C07270=1079.126,-46.331,-56.939,173.614,20.204,153.491
C07271=1079.132,-46.080,-56.951,173.616,20.206,153.491
C07272=1079.137,-45.831,-56.963,173.617,20.207,153.491
C07273=1079.144,-45.582,-56.975,173.618,20.209,153.491
C07274=1079.150,-45.332,-56.987,173.621,20.212,153.491
C07275=1079.155,-45.083,-57.000,173.622,20.214,153.492
C07276=1079.162,-44.833,-57.012,173.623,20.215,153.492
C07277=1079.168,-44.583,-57.024,173.625,20.217,153.492
C07278=1079.173,-44.334,-57.035,173.626,20.219,153.492
C07279=1079.179,-44.084,-57.048,173.627,20.221,153.492
C07280=1079.185,-43.834,-57.060,173.629,20.223,153.492
C07281=1079.192,-43.584,-57.072,173.630,20.225,153.492
C07282=1079.197,-43.335,-57.084,173.632,20.227,153.492
C07283=1079.203,-43.085,-57.097,173.633,20.229,153.493
C07284=1079.210,-42.836,-57.109,173.635,20.230,153.493
C07285=1079.215,-42.586,-57.121,173.636,20.232,153.493
C07286=1079.221,-42.337,-57.134,173.637,20.234,153.493
C07287=1079.228,-42.087,-57.146,173.639,20.236,153.493
C07288=1079.233,-41.837,-57.158,173.640,20.238,153.493
C07289=1079.239,-41.588,-57.170,173.642,20.240,153.493
C07290=1079.245,-41.338,-57.183,173.644,20.242,153.493
C07291=1079.251,-41.088,-57.195,173.645,20.244,153.494
C07292=1079.257,-40.839,-57.207,173.646,20.246,153.494
C07293=1079.263,-40.589,-57.220,173.648,20.248,153.494
C07294=1079.269,-40.340,-57.231,173.649,20.250,153.494
C07295=1079.275,-40.090,-57.244,173.650,20.252,153.494
C07296=1079.281,-39.840,-57.257,173.652,20.253,153.494
C07297=1079.288,-39.590,-57.269,173.653,20.255,153.494
C07298=1079.293,-39.341,-57.281,173.655,20.258,153.494
C07299=1079.299,-39.091,-57.293,173.657,20.260,153.495
C07300=1079.305,-38.842,-57.306,173.658,20.262,153.495
C07301=1079.311,-38.592,-57.318,173.659,20.263,153.495
C07302=1079.317,-38.342,-57.330,173.661,20.265,153.495
C07303=1079.323,-38.093,-57.343,173.662,20.267,153.495
C07304=1079.329,-37.843,-57.355,173.663,20.269,153.495
C07305=1079.334,-37.593,-57.368,173.665,20.272,153.495
C07306=1079.340,-37.343,-57.380,173.667,20.274,153.496
C07307=1079.346,-37.094,-57.392,173.668,20.276,153.496
C07308=1079.353,-36.845,-57.405,173.669,20.278,153.496
C07309=1079.359,-36.595,-57.418,173.671,20.279,153.496
C07310=1079.364,-36.345,-57.430,173.672,20.281,153.496
C07311=1079.370,-36.096,-57.442,173.673,20.283,153.496
C07312=1079.376,-35.846,-57.455,173.674,20.285,153.496
C07313=1079.382,-35.596,-57.467,173.677,20.288,153.497
C07314=1079.388,-35.347,-57.480,173.678,20.290,153.497
C07315=1079.393,-35.097,-57.493,173.679,20.292,153.497
C07316=1079.399,-34.848,-57.505,173.680,20.294,153.497
C07317=1079.406,-34.599,-57.517,173.682,20.296,153.497
C07318=1079.412,-34.349,-57.530,173.683,20.298,153.497
C07319=1079.417,-34.099,-57.543,173.685,20.300,153.497
C07320=1079.423,-33.849,-57.555,173.687,20.302,153.498
C07321=1079.430,-33.575,-57.569,173.688,20.304,153.498
C07322=1079.436,-33.302,-57.583,173.689,20.306,153.498
C07323=1079.442,-33.028,-57.596,173.691,20.309,153.498
C07324=1079.449,-32.754,-57.610,173.692,20.311,153.498
C07325=1079.455,-32.504,-57.624,173.694,20.313,153.499
C07326=1079.461,-32.254,-57.636,173.695,20.315,153.499
C07327=1079.467,-32.004,-57.649,173.697,20.317,153.499
C07328=1079.473,-31.755,-57.661,173.699,20.318,153.499
C07329=1079.479,-31.505,-57.675,173.700,20.320,153.499
C07330=1079.484,-31.256,-57.687,173.701,20.322,153.499
C07331=1079.491,-31.007,-57.699,173.703,20.324,153.499
C07332=1079.497,-30.757,-57.712,173.704,20.326,153.500
C07333=1079.503,-30.507,-57.725,173.705,20.328,153.500
C07334=1079.509,-30.258,-57.737,173.707,20.331,153.500
C07335=1079.515,-30.008,-57.750,173.709,20.333,153.500
C07336=1079.521,-29.758,-57.763,173.710,20.335,153.500
C07337=1079.527,-29.509,-57.775,173.711,20.337,153.500
C07338=1079.532,-29.259,-57.788,173.712,20.339,153.500
C07339=1079.538,-29.010,-57.801,173.714,20.341,153.501
C07340=1079.544,-28.760,-57.813,173.716,20.343,153.501
C07341=1079.550,-28.510,-57.826,173.717,20.345,153.501
C07342=1079.556,-28.261,-57.839,173.719,20.347,153.501
C07343=1079.562,-28.011,-57.852,173.720,20.349,153.501
C07344=1079.568,-27.761,-57.864,173.721,20.351,153.501
C07345=1079.574,-27.512,-57.878,173.722,20.353,153.501
C07346=1079.580,-27.262,-57.890,173.725,20.355,153.502
C07347=1079.587,-27.013,-57.903,173.726,20.357,153.502
C07348=1079.592,-26.763,-57.916,173.727,20.359,153.502
C07349=1079.598,-26.513,-57.929,173.728,20.361,153.502
C07350=1079.604,-26.264,-57.942,173.730,20.363,153.502
C07351=1079.609,-26.014,-57.955,173.731,20.365,153.502
C07352=1079.615,-25.765,-57.968,173.733,20.368,153.503
C07353=1079.621,-25.515,-57.980,173.734,20.370,153.503
C07354=1079.627,-25.266,-57.994,173.736,20.372,153.503
C07355=1079.633,-25.016,-58.006,173.737,20.374,153.503
C07356=1079.639,-24.766,-58.019,173.738,20.376,153.503
C07357=1079.645,-24.517,-58.033,173.739,20.378,153.504
C07358=1079.651,-24.267,-58.045,173.742,20.381,153.504
C07359=1079.657,-24.017,-58.059,173.743,20.383,153.504
C07360=1079.663,-23.768,-58.071,173.744,20.385,153.504
C07361=1079.668,-23.518,-58.085,173.745,20.387,153.504
C07362=1079.674,-23.268,-58.097,173.747,20.389,153.504
C07363=1079.680,-23.020,-58.110,173.748,20.391,153.504
C07364=1079.686,-22.770,-58.123,173.750,20.393,153.505
C07365=1079.692,-22.520,-58.136,173.751,20.395,153.505
C07366=1079.697,-22.270,-58.149,173.753,20.397,153.505
C07367=1079.703,-22.021,-58.163,173.754,20.399,153.505
C07368=1079.709,-21.771,-58.175,173.755,20.401,153.505
C07369=1079.715,-21.522,-58.188,173.757,20.403,153.505
C07370=1079.722,-21.273,-58.202,173.759,20.405,153.506
C07371=1079.727,-21.022,-58.215,173.760,20.407,153.506
C07372=1079.733,-20.773,-58.228,173.761,20.409,153.506
C07373=1079.739,-20.523,-58.241,173.763,20.411,153.506
C07374=1079.745,-20.274,-58.254,173.764,20.413,153.506
C07375=1079.751,-20.024,-58.268,173.766,20.416,153.507
C07376=1079.757,-19.774,-58.280,173.767,20.418,153.507
C07377=1079.763,-19.525,-58.294,173.768,20.420,153.507
C07378=1079.769,-19.275,-58.306,173.770,20.422,153.507
C07379=1079.774,-19.026,-58.320,173.771,20.424,153.507
C07380=1079.780,-18.776,-58.333,173.772,20.426,153.507
C07381=1079.786,-18.527,-58.346,173.774,20.429,153.507
C07382=1079.792,-18.277,-58.359,173.776,20.431,153.508
C07383=1079.798,-18.028,-58.373,173.777,20.433,153.508
C07384=1079.804,-17.778,-58.386,173.778,20.435,153.508
C07385=1079.811,-17.503,-58.400,173.780,20.437,153.508
C07386=1079.817,-17.228,-58.415,173.782,20.440,153.508
C07387=1079.824,-16.953,-58.430,173.783,20.442,153.509
C07388=1079.830,-16.679,-58.443,173.785,20.444,153.509
C07389=1079.837,-16.429,-58.457,173.786,20.446,153.509
C07390=1079.842,-16.180,-58.471,173.788,20.448,153.509
C07391=1079.849,-15.930,-58.484,173.789,20.450,153.509
C07392=1079.854,-15.680,-58.497,173.791,20.453,153.509
C07393=1079.860,-15.431,-58.511,173.792,20.455,153.510
C07394=1079.866,-15.182,-58.524,173.793,20.457,153.510
C07395=1079.872,-14.932,-58.537,173.795,20.459,153.510
C07396=1079.878,-14.682,-58.550,173.796,20.461,153.510
C07397=1079.884,-14.433,-58.564,173.797,20.463,153.510
C07398=1079.889,-14.183,-58.577,173.799,20.465,153.510
C07399=1079.895,-13.934,-58.591,173.800,20.468,153.511
C07400=1079.901,-13.684,-58.604,173.802,20.470,153.511
C07401=1079.907,-13.435,-58.617,173.803,20.472,153.511
C07402=1079.913,-13.185,-58.630,173.804,20.474,153.511
C07403=1079.919,-12.936,-58.644,173.806,20.476,153.511
C07404=1079.925,-12.686,-58.658,173.808,20.478,153.512
C07405=1079.930,-12.436,-58.671,173.809,20.481,153.512
C07406=1079.936,-12.187,-58.684,173.810,20.483,153.512
C07407=1079.942,-11.937,-58.698,173.811,20.485,153.512
C07408=1079.948,-11.687,-58.711,173.814,20.487,153.512
C07409=1079.954,-11.438,-58.725,173.815,20.489,153.512
C07410=1079.960,-11.189,-58.739,173.816,20.491,153.513
C07411=1079.965,-10.938,-58.752,173.817,20.494,153.513
C07412=1079.972,-10.689,-58.765,173.819,20.496,153.513
C07413=1079.977,-10.440,-58.779,173.821,20.498,153.513
C07414=1079.983,-10.190,-58.792,173.822,20.500,153.513
C07415=1079.989,-9.941,-58.806,173.823,20.502,153.514
C07416=1079.995,-9.691,-58.819,173.825,20.504,153.514
C07417=1080.001,-9.441,-58.834,173.826,20.507,153.514
C07418=1080.007,-9.192,-58.847,173.828,20.509,153.514
C07419=1080.013,-8.942,-58.861,173.829,20.511,153.514
C07420=1080.019,-8.693,-58.874,173.830,20.513,153.515
C07421=1080.024,-8.443,-58.887,173.832,20.515,153.515
C07422=1080.030,-8.193,-58.901,173.833,20.517,153.515
C07423=1080.036,-7.944,-58.914,173.835,20.520,153.515
C07424=1080.042,-7.694,-58.928,173.836,20.522,153.515
C07425=1080.048,-7.445,-58.942,173.837,20.524,153.515
C07426=1080.053,-7.195,-58.956,173.839,20.526,153.516
C07427=1080.060,-6.946,-58.969,173.840,20.528,153.516
C07428=1080.065,-6.696,-58.983,173.842,20.530,153.516
C07429=1080.071,-6.447,-58.996,173.843,20.533,153.516
C07430=1080.077,-6.197,-59.010,173.845,20.535,153.516
C07431=1080.084,-5.947,-59.024,173.846,20.537,153.517
C07432=1080.089,-5.698,-59.037,173.848,20.539,153.517
C07433=1080.095,-5.448,-59.051,173.849,20.541,153.517
C07434=1080.101,-5.199,-59.064,173.850,20.544,153.517
C07435=1080.107,-4.949,-59.079,173.852,20.546,153.517
C07436=1080.113,-4.699,-59.092,173.853,20.548,153.517
C07437=1080.119,-4.450,-59.106,173.855,20.550,153.518
C07438=1080.125,-4.201,-59.120,173.856,20.552,153.518
C07439=1080.131,-3.952,-59.134,173.858,20.554,153.518
C07440=1080.137,-3.701,-59.148,173.859,20.557,153.518
C07441=1080.143,-3.452,-59.161,173.860,20.559,153.518
C07442=1080.148,-3.202,-59.175,173.862,20.561,153.519
C07443=1080.154,-2.953,-59.189,173.864,20.563,153.519
C07444=1080.160,-2.704,-59.202,173.865,20.566,153.519
C07445=1080.166,-2.453,-59.216,173.866,20.568,153.519
C07446=1080.172,-2.204,-59.230,173.868,20.570,153.519
C07447=1080.177,-1.954,-59.244,173.869,20.572,153.519
C07448=1080.183,-1.705,-59.259,173.871,20.575,153.520
C07449=1080.190,-1.429,-59.273,173.872,20.577,153.520
C07450=1080.196,-1.153,-59.289,173.874,20.580,153.520
C07451=1080.202,-0.875,-59.305,173.875,20.582,153.520
C07452=1080.209,-0.600,-59.320,173.877,20.585,153.521
C07453=1080.215,-0.350,-59.334,173.878,20.587,153.521
C07454=1080.220,-0.100,-59.348,173.880,20.589,153.521
C07455=1080.226,0.148,-59.362,173.881,20.591,153.521
C07456=1080.232,0.399,-59.376,173.883,20.593,153.521
C07457=1080.237,0.648,-59.390,173.884,20.595,153.522
C07458=1080.244,0.898,-59.403,173.885,20.598,153.522
C07459=1080.249,1.147,-59.417,173.887,20.600,153.522
C07460=1080.255,1.396,-59.432,173.889,20.602,153.522
C07461=1080.261,1.646,-59.446,173.890,20.604,153.522
C07462=1080.266,1.896,-59.460,173.891,20.607,153.523
C07463=1080.272,2.146,-59.474,173.892,20.609,153.523
C07464=1080.278,2.395,-59.488,173.894,20.611,153.523
C07465=1080.284,2.644,-59.502,173.896,20.614,153.523
C07466=1080.290,2.894,-59.516,173.897,20.616,153.523
C07467=1080.296,3.143,-59.531,173.898,20.618,153.524
C07468=1080.301,3.393,-59.544,173.900,20.620,153.524
C07469=1080.307,3.643,-59.559,173.901,20.623,153.524
C07470=1080.313,3.892,-59.572,173.903,20.625,153.524
C07471=1080.319,4.141,-59.587,173.904,20.627,153.524
C07472=1080.324,4.391,-59.601,173.905,20.629,153.525
C07473=1080.331,4.641,-59.615,173.907,20.632,153.525
C07474=1080.337,4.890,-59.629,173.909,20.634,153.525
C07475=1080.342,5.139,-59.643,173.910,20.636,153.525
C07476=1080.348,5.390,-59.657,173.911,20.638,153.525
C07477=1080.354,5.639,-59.672,173.913,20.641,153.526
C07478=1080.359,5.888,-59.686,173.914,20.643,153.526
C07479=1080.366,6.138,-59.701,173.916,20.644,153.526
C07480=1080.371,6.388,-59.714,173.917,20.647,153.526
C07481=1080.377,6.637,-59.728,173.918,20.649,153.526
C07482=1080.383,6.887,-59.743,173.920,20.651,153.527
C07483=1080.389,7.136,-59.757,173.921,20.654,153.527
C07484=1080.395,7.385,-59.771,173.923,20.656,153.527
C07485=1080.401,7.635,-59.785,173.924,20.658,153.527
C07486=1080.407,7.885,-59.799,173.926,20.660,153.527
C07487=1080.413,8.134,-59.814,173.927,20.663,153.528
C07488=1080.419,8.384,-59.828,173.929,20.665,153.528
C07489=1080.424,8.633,-59.843,173.930,20.667,153.528
C07490=1080.430,8.883,-59.856,173.932,20.669,153.528
C07491=1080.436,9.132,-59.871,173.933,20.672,153.528
C07492=1080.442,9.382,-59.885,173.934,20.674,153.529
C07493=1080.447,9.631,-59.900,173.936,20.676,153.529
C07494=1080.454,9.881,-59.914,173.938,20.678,153.529
C07495=1080.459,10.130,-59.929,173.939,20.681,153.529
C07496=1080.465,10.380,-59.943,173.940,20.683,153.529
C07497=1080.471,10.629,-59.958,173.942,20.685,153.530
C07498=1080.477,10.879,-59.971,173.944,20.687,153.530
C07499=1080.483,11.128,-59.986,173.945,20.690,153.530
C07500=1080.489,11.378,-60.000,173.946,20.691,153.530
C07501=1080.496,11.627,-60.015,173.947,20.693,153.530
C07502=1080.501,11.877,-60.028,173.949,20.695,153.530
C07503=1080.508,12.127,-60.043,173.951,20.698,153.531
C07504=1080.513,12.376,-60.057,173.952,20.700,153.531
C07505=1080.519,12.625,-60.072,173.953,20.702,153.531
C07506=1080.525,12.875,-60.087,173.955,20.704,153.531
C07507=1080.531,13.124,-60.101,173.957,20.707,153.532
C07508=1080.537,13.374,-60.116,173.958,20.709,153.532
C07509=1080.542,13.624,-60.129,173.959,20.711,153.532
C07510=1080.549,13.873,-60.144,173.960,20.713,153.532
C07511=1080.555,14.122,-60.159,173.962,20.716,153.532
C07512=1080.561,14.372,-60.173,173.964,20.718,153.532
C07513=1080.566,14.650,-60.189,173.965,20.720,153.533
C07514=1080.573,14.929,-60.206,173.967,20.723,153.533
C07515=1080.579,15.207,-60.222,173.969,20.726,153.533
C07516=1080.586,15.485,-60.238,173.970,20.728,153.533
C07517=1080.592,15.735,-60.253,173.971,20.731,153.534
C07518=1080.598,15.984,-60.268,173.974,20.733,153.534
C07519=1080.604,16.234,-60.282,173.975,20.735,153.534
C07520=1080.610,16.483,-60.297,173.976,20.737,153.534
C07521=1080.615,16.732,-60.311,173.977,20.739,153.534
C07522=1080.621,16.983,-60.326,173.979,20.742,153.535
C07523=1080.626,17.232,-60.341,173.980,20.744,153.535
C07524=1080.633,17.482,-60.356,173.982,20.746,153.535
C07525=1080.639,17.730,-60.370,173.983,20.748,153.535
C07526=1080.645,17.981,-60.385,173.985,20.751,153.535
C07527=1080.650,18.230,-60.400,173.986,20.753,153.536
C07528=1080.656,18.480,-60.415,173.988,20.755,153.536
C07529=1080.662,18.729,-60.429,173.989,20.757,153.536
C07530=1080.668,18.979,-60.444,173.991,20.760,153.536
C07531=1080.674,19.228,-60.458,173.992,20.762,153.536
C07532=1080.679,19.478,-60.474,173.994,20.764,153.537
C07533=1080.685,19.727,-60.488,173.995,20.767,153.537
C07534=1080.692,19.976,-60.503,173.997,20.769,153.537
C07535=1080.697,20.226,-60.517,173.998,20.771,153.537
C07536=1080.703,20.476,-60.533,173.999,20.773,153.537
C07537=1080.708,20.725,-60.547,174.001,20.776,153.538
C07538=1080.714,20.974,-60.562,174.003,20.778,153.538
C07539=1080.720,21.224,-60.577,174.004,20.780,153.538
C07540=1080.725,21.473,-60.591,174.005,20.782,153.538
C07541=1080.732,21.723,-60.606,174.007,20.785,153.538
C07542=1080.737,21.972,-60.621,174.008,20.787,153.539
C07543=1080.743,22.222,-60.636,174.010,20.789,153.539
C07544=1080.749,22.471,-60.651,174.011,20.791,153.539
C07545=1080.755,22.721,-60.666,174.013,20.794,153.539
C07546=1080.760,22.970,-60.681,174.014,20.796,153.539
C07547=1080.767,23.220,-60.696,174.016,20.798,153.540
C07548=1080.772,23.470,-60.711,174.017,20.801,153.540
C07549=1080.778,23.719,-60.725,174.019,20.803,153.540
C07550=1080.784,23.969,-60.740,174.020,20.805,153.540
C07551=1080.789,24.218,-60.755,174.021,20.808,153.541
C07552=1080.796,24.468,-60.770,174.023,20.810,153.541
C07553=1080.801,24.717,-60.785,174.025,20.812,153.541
C07554=1080.807,24.967,-60.800,174.026,20.814,153.541
C07555=1080.813,25.216,-60.815,174.027,20.816,153.541
C07556=1080.819,25.466,-60.831,174.029,20.819,153.541
C07557=1080.824,25.714,-60.845,174.031,20.821,153.542
C07558=1080.831,25.964,-60.860,174.032,20.823,153.542
C07559=1080.836,26.214,-60.876,174.034,20.826,153.542
C07560=1080.842,26.463,-60.890,174.035,20.828,153.542
C07561=1080.849,26.713,-60.905,174.036,20.830,153.543
C07562=1080.854,26.962,-60.920,174.038,20.832,153.543
C07563=1080.860,27.212,-60.935,174.040,20.835,153.543
C07564=1080.866,27.462,-60.951,174.041,20.837,153.543
C07565=1080.871,27.711,-60.965,174.042,20.839,153.543
C07566=1080.877,27.961,-60.981,174.043,20.841,153.544
C07567=1080.883,28.209,-60.996,174.045,20.844,153.544
C07568=1080.889,28.459,-61.010,174.047,20.846,153.544
C07569=1080.895,28.708,-61.026,174.048,20.848,153.544
C07570=1080.901,28.957,-61.041,174.050,20.850,153.544
C07571=1080.907,29.207,-61.057,174.051,20.853,153.545
C07572=1080.912,29.457,-61.072,174.053,20.855,153.545
C07573=1080.918,29.706,-61.087,174.054,20.857,153.545
C07574=1080.923,29.956,-61.102,174.056,20.860,153.545
C07575=1080.929,30.205,-61.117,174.057,20.862,153.545
C07576=1080.935,30.455,-61.133,174.058,20.864,153.546
C07577=1080.941,30.735,-61.150,174.061,20.867,153.546
C07578=1080.948,31.014,-61.167,174.063,20.870,153.546
C07579=1080.954,31.294,-61.184,174.064,20.872,153.546
C07580=1080.961,31.574,-61.201,174.066,20.874,153.546
C07581=1080.967,31.823,-61.216,174.067,20.876,153.547
C07582=1080.972,32.073,-61.231,174.068,20.879,153.547
C07583=1080.978,32.321,-61.247,174.070,20.881,153.547
C07584=1080.984,32.571,-61.262,174.072,20.883,153.547
C07585=1080.990,32.821,-61.278,174.073,20.886,153.548
C07586=1080.995,33.070,-61.292,174.074,20.888,153.548
C07587=1081.001,33.320,-61.308,174.076,20.890,153.548
C07588=1081.008,33.569,-61.324,174.077,20.893,153.548
C07589=1081.013,33.818,-61.339,174.079,20.895,153.548
C07590=1081.019,34.068,-61.354,174.081,20.897,153.548
C07591=1081.025,34.318,-61.369,174.082,20.900,153.549
C07592=1081.030,34.567,-61.385,174.083,20.902,153.549
C07593=1081.037,34.816,-61.400,174.085,20.904,153.549
C07594=1081.042,35.066,-61.416,174.087,20.906,153.549
C07595=1081.048,35.315,-61.432,174.088,20.908,153.550
C07596=1081.054,35.565,-61.446,174.089,20.910,153.550
C07597=1081.060,35.815,-61.462,174.091,20.913,153.550
C07598=1081.065,36.064,-61.477,174.093,20.915,153.550
C07599=1081.071,36.313,-61.493,174.094,20.917,153.550
C07600=1081.077,36.563,-61.508,174.096,20.920,153.550
C07601=1081.083,36.813,-61.524,174.097,20.922,153.551
C07602=1081.089,37.061,-61.539,174.098,20.924,153.551
C07603=1081.094,37.311,-61.555,174.101,20.927,153.551
C07604=1081.100,37.561,-61.570,174.102,20.929,153.551
C07605=1081.106,37.810,-61.586,174.103,20.931,153.552
C07606=1081.112,38.059,-61.601,174.104,20.933,153.552
C07607=1081.118,38.309,-61.617,174.106,20.936,153.552
C07608=1081.123,38.559,-61.633,174.108,20.938,153.552
C07609=1081.129,38.808,-61.648,174.109,20.940,153.552
C07610=1081.135,39.057,-61.664,174.111,20.943,153.553
C07611=1081.141,39.307,-61.679,174.112,20.945,153.553
C07612=1081.146,39.556,-61.695,174.114,20.947,153.553
C07613=1081.152,39.806,-61.711,174.116,20.950,153.553
C07614=1081.158,40.055,-61.726,174.117,20.952,153.553
C07615=1081.163,40.304,-61.742,174.118,20.954,153.554
C07616=1081.169,40.554,-61.757,174.120,20.957,153.554
C07617=1081.175,40.803,-61.773,174.121,20.959,153.554
C07618=1081.181,41.053,-61.789,174.123,20.960,153.554
C07619=1081.186,41.302,-61.805,174.125,20.963,153.554
C07620=1081.192,41.552,-61.820,174.126,20.965,153.555
C07621=1081.198,41.801,-61.836,174.127,20.967,153.555
C07622=1081.204,42.051,-61.852,174.129,20.970,153.555
C07623=1081.209,42.300,-61.867,174.131,20.972,153.555
C07624=1081.215,42.550,-61.883,174.132,20.974,153.555
C07625=1081.221,42.799,-61.899,174.134,20.977,153.556
C07626=1081.227,43.049,-61.914,174.135,20.979,153.556
C07627=1081.233,43.298,-61.930,174.137,20.981,153.556
C07628=1081.238,43.547,-61.946,174.138,20.983,153.556
C07629=1081.244,43.796,-61.962,174.140,20.986,153.556
C07630=1081.250,44.046,-61.977,174.141,20.988,153.557
C07631=1081.256,44.296,-61.994,174.143,20.990,153.557
C07632=1081.261,44.544,-62.010,174.145,20.993,153.557
C07633=1081.267,44.794,-62.025,174.146,20.995,153.557
C07634=1081.273,45.044,-62.041,174.147,20.997,153.558
C07635=1081.278,45.293,-62.057,174.149,21.000,153.558
C07636=1081.284,45.542,-62.073,174.150,21.002,153.558
C07637=1081.290,45.792,-62.089,174.152,21.004,153.558
C07638=1081.295,46.042,-62.105,174.154,21.007,153.558
C07639=1081.301,46.291,-62.121,174.155,21.009,153.558
C07640=1081.306,46.540,-62.136,174.156,21.011,153.559
C07641=1081.313,46.820,-62.155,174.158,21.013,153.559
C07642=1081.319,47.100,-62.172,174.160,21.016,153.559
C07643=1081.326,47.380,-62.190,174.161,21.019,153.559
C07644=1081.331,47.660,-62.208,174.164,21.021,153.560
C07645=1081.337,47.909,-62.224,174.165,21.024,153.560
C07646=1081.343,48.158,-62.241,174.167,21.026,153.560
C07647=1081.349,48.408,-62.256,174.168,21.028,153.560
C07648=1081.354,48.657,-62.272,174.169,21.031,153.561
C07649=1081.360,48.906,-62.288,174.172,21.033,153.561
C07650=1081.366,49.156,-62.305,174.173,21.035,153.561
C07651=1081.372,49.406,-62.320,174.174,21.037,153.561
C07652=1081.378,49.655,-62.336,174.176,21.040,153.561
C07653=1081.384,49.904,-62.353,174.178,21.042,153.561
C07654=1081.389,50.153,-62.369,174.179,21.044,153.562
C07655=1081.394,50.403,-62.385,174.181,21.047,153.562
C07656=1081.400,50.653,-62.401,174.182,21.049,153.562
C07657=1081.406,50.902,-62.417,174.183,21.051,153.562
C07658=1081.412,51.151,-62.434,174.185,21.054,153.562
C07659=1081.418,51.401,-62.450,174.187,21.056,153.563
C07660=1081.423,51.651,-62.465,174.188,21.057,153.563
C07661=1081.429,51.899,-62.481,174.190,21.060,153.563
C07662=1081.435,52.149,-62.497,174.191,21.062,153.563
C07663=1081.441,52.398,-62.514,174.193,21.064,153.563
C07664=1081.446,52.648,-62.531,174.195,21.067,153.564
C07665=1081.451,52.898,-62.546,174.196,21.069,153.564
C07666=1081.457,53.147,-62.562,174.198,21.072,153.564
C07667=1081.463,53.396,-62.579,174.200,21.074,153.564
C07668=1081.469,53.646,-62.595,174.201,21.076,153.565
C07669=1081.475,53.895,-62.611,174.203,21.078,153.565
C07670=1081.481,54.144,-62.627,174.204,21.080,153.565
C07671=1081.486,54.393,-62.644,174.205,21.083,153.565
C07672=1081.492,54.643,-62.660,174.208,21.085,153.565
C07673=1081.498,54.892,-62.676,174.209,21.087,153.565
C07674=1081.503,55.142,-62.692,174.210,21.089,153.566
C07675=1081.509,55.391,-62.708,174.212,21.092,153.566
C07676=1081.515,55.641,-62.724,174.213,21.094,153.566
C07677=1081.520,55.890,-62.741,174.215,21.096,153.566
C07678=1081.526,56.140,-62.758,174.217,21.098,153.566
C07679=1081.532,56.389,-62.774,174.218,21.100,153.567
C07680=1081.538,56.638,-62.790,174.220,21.103,153.567
C07681=1081.544,56.888,-62.806,174.222,21.105,153.567
C07682=1081.550,57.137,-62.823,174.223,21.107,153.567
C07683=1081.555,57.387,-62.839,174.225,21.110,153.567
C07684=1081.561,57.636,-62.856,174.226,21.112,153.568
C07685=1081.567,57.885,-62.872,174.228,21.114,153.568
C07686=1081.573,58.135,-62.888,174.230,21.117,153.568
C07687=1081.579,58.384,-62.905,174.231,21.118,153.568
C07688=1081.584,58.634,-62.921,174.232,21.120,153.568
C07689=1081.590,58.883,-62.938,174.235,21.123,153.568
C07690=1081.596,59.132,-62.954,174.236,21.125,153.569
C07691=1081.602,59.382,-62.970,174.238,21.128,153.569
C07692=1081.608,59.631,-62.987,174.239,21.130,153.569
C07693=1081.614,59.880,-63.004,174.241,21.132,153.569
C07694=1081.620,60.129,-63.020,174.243,21.134,153.569
C07695=1081.626,60.379,-63.036,174.244,21.137,153.570
C07696=1081.631,60.628,-63.053,174.245,21.138,153.570
C07697=1081.637,60.878,-63.070,174.247,21.141,153.570
C07698=1081.643,61.127,-63.086,174.249,21.143,153.570
C07699=1081.649,61.377,-63.102,174.250,21.145,153.570
C07700=1081.654,61.626,-63.119,174.252,21.147,153.570
C07701=1081.660,61.876,-63.135,174.254,21.149,153.571
C07702=1081.666,62.124,-63.152,174.256,21.152,153.571
C07703=1081.672,62.374,-63.168,174.257,21.154,153.571
C07704=1081.677,62.623,-63.185,174.258,21.156,153.571
C07705=1081.684,62.903,-63.204,174.261,21.158,153.571
C07706=1081.692,63.182,-63.222,174.262,21.161,153.572
C07707=1081.698,63.462,-63.241,174.264,21.163,153.572
C07708=1081.704,63.741,-63.259,174.266,21.166,153.572
C07709=1081.710,63.991,-63.276,174.267,21.168,153.572
C07710=1081.716,64.240,-63.292,174.269,21.171,153.572
C07711=1081.722,64.490,-63.309,174.271,21.172,153.572
C07712=1081.728,64.739,-63.327,174.273,21.175,153.573
C07713=1081.734,64.988,-63.343,174.274,21.177,153.573
C07714=1081.739,65.238,-63.360,174.276,21.179,153.573
C07715=1081.745,65.487,-63.376,174.278,21.182,153.573
C07716=1081.750,65.737,-63.394,174.279,21.184,153.573
C07717=1081.756,65.986,-63.410,174.280,21.186,153.574
C07718=1081.762,66.235,-63.426,174.282,21.188,153.574
C07719=1081.767,66.485,-63.443,174.284,21.190,153.574
C07720=1081.774,66.734,-63.460,174.286,21.192,153.574
C07721=1081.779,66.983,-63.477,174.287,21.195,153.574
C07722=1081.785,67.233,-63.493,174.288,21.197,153.575
C07723=1081.790,67.482,-63.511,174.291,21.199,153.575
C07724=1081.797,67.732,-63.527,174.292,21.201,153.575
C07725=1081.802,67.981,-63.544,174.294,21.204,153.575
C07726=1081.808,68.230,-63.561,174.295,21.206,153.575
C07727=1081.814,68.480,-63.578,174.297,21.208,153.575
C07728=1081.819,68.729,-63.595,174.299,21.210,153.576
C07729=1081.825,68.978,-63.612,174.300,21.212,153.576
C07730=1081.830,69.228,-63.629,174.302,21.215,153.576
C07731=1081.837,69.477,-63.646,174.304,21.217,153.576
C07732=1081.842,69.726,-63.662,174.305,21.219,153.576
C07733=1081.848,69.976,-63.679,174.307,21.222,153.577
C07734=1081.854,70.225,-63.697,174.308,21.223,153.577
C07735=1081.860,70.475,-63.713,174.311,21.226,153.577
C07736=1081.865,70.724,-63.730,174.312,21.228,153.577
C07737=1081.871,70.973,-63.747,174.313,21.230,153.577
C07738=1081.877,71.222,-63.764,174.315,21.232,153.577
C07739=1081.882,71.472,-63.781,174.317,21.235,153.578
C07740=1081.887,71.721,-63.799,174.319,21.237,153.578
C07741=1081.894,71.971,-63.815,174.320,21.239,153.578
C07742=1081.900,72.220,-63.833,174.321,21.241,153.578
C07743=1081.905,72.470,-63.850,174.324,21.243,153.578
C07744=1081.911,72.718,-63.867,174.325,21.245,153.578
C07745=1081.916,72.968,-63.884,174.327,21.248,153.579
C07746=1081.922,73.217,-63.901,174.328,21.250,153.579
C07747=1081.928,73.466,-63.917,174.330,21.252,153.579
C07748=1081.934,73.716,-63.935,174.332,21.255,153.579
C07749=1081.939,73.966,-63.952,174.333,21.256,153.579
C07750=1081.945,74.214,-63.969,174.335,21.259,153.579
C07751=1081.951,74.464,-63.986,174.337,21.261,153.580
C07752=1081.956,74.713,-64.004,174.339,21.263,153.580
C07753=1081.962,74.963,-64.021,174.340,21.266,153.580
C07754=1081.968,75.212,-64.038,174.341,21.268,153.580
C07755=1081.974,75.461,-64.055,174.344,21.270,153.580
C07756=1081.979,75.711,-64.072,174.345,21.272,153.581
C07757=1081.985,75.960,-64.089,174.347,21.274,153.581
C07758=1081.991,76.210,-64.106,174.348,21.276,153.581
C07759=1081.996,76.459,-64.124,174.350,21.278,153.581
C07760=1082.002,76.708,-64.141,174.352,21.281,153.581
C07761=1082.008,76.957,-64.158,174.353,21.283,153.581
C07762=1082.013,77.206,-64.175,174.356,21.285,153.581
C07763=1082.020,77.456,-64.193,174.357,21.287,153.582
C07764=1082.025,77.706,-64.210,174.359,21.290,153.582
C07765=1082.031,77.955,-64.227,174.360,21.292,153.582
C07766=1082.037,78.204,-64.245,174.362,21.294,153.582
C07767=1082.042,78.454,-64.262,174.364,21.296,153.582
C07768=1082.048,78.703,-64.279,174.365,21.298,153.583
C07769=1082.055,78.982,-64.299,174.367,21.300,153.583
C07770=1082.061,79.262,-64.318,174.369,21.303,153.583
C07771=1082.067,79.541,-64.338,174.371,21.305,153.583
C07772=1082.073,79.821,-64.357,174.373,21.308,153.583
C07773=1082.079,80.070,-64.374,174.375,21.311,153.584
C07774=1082.085,80.319,-64.392,174.376,21.313,153.584
C07775=1082.091,80.568,-64.410,174.378,21.315,153.584
C07776=1082.096,80.818,-64.427,174.380,21.317,153.584
C07777=1082.101,81.067,-64.444,174.381,21.319,153.584
C07778=1082.107,81.317,-64.462,174.383,21.321,153.584
C07779=1082.113,81.566,-64.480,174.385,21.323,153.585
C07780=1082.118,81.815,-64.497,174.387,21.326,153.585
C07781=1082.124,82.065,-64.514,174.388,21.328,153.585
C07782=1082.130,82.314,-64.532,174.390,21.330,153.585
C07783=1082.135,82.563,-64.550,174.392,21.332,153.585
C07784=1082.141,82.812,-64.567,174.393,21.334,153.585
C07785=1082.147,83.062,-64.585,174.395,21.337,153.586
C07786=1082.152,83.311,-64.603,174.396,21.339,153.586
C07787=1082.158,83.561,-64.620,174.399,21.341,153.586
C07788=1082.163,83.810,-64.637,174.400,21.343,153.586
C07789=1082.169,84.060,-64.655,174.402,21.345,153.586
C07790=1082.176,84.308,-64.672,174.403,21.347,153.586
C07791=1082.181,84.557,-64.690,174.406,21.350,153.587
C07792=1082.187,84.807,-64.708,174.407,21.352,153.587
C07793=1082.193,85.056,-64.725,174.408,21.354,153.587
C07794=1082.198,85.305,-64.743,174.411,21.356,153.587
C07795=1082.204,85.555,-64.761,174.412,21.358,153.587
C07796=1082.210,85.804,-64.778,174.414,21.360,153.587
C07797=1082.215,86.053,-64.796,174.415,21.362,153.588
C07798=1082.221,86.303,-64.814,174.418,21.365,153.588
C07799=1082.227,86.552,-64.831,174.419,21.367,153.588
C07800=1082.233,86.801,-64.849,174.421,21.369,153.588
C07801=1082.238,87.051,-64.867,174.423,21.371,153.588
C07802=1082.243,87.300,-64.885,174.425,21.373,153.588
C07803=1082.249,87.549,-64.902,174.426,21.375,153.588
C07804=1082.255,87.799,-64.920,174.428,21.378,153.589
C07805=1082.261,88.048,-64.938,174.430,21.380,153.589
C07806=1082.267,88.297,-64.956,174.431,21.382,153.589
C07807=1082.272,88.546,-64.973,174.433,21.384,153.589
C07808=1082.278,88.796,-64.991,174.435,21.386,153.589
C07809=1082.284,89.045,-65.009,174.437,21.388,153.589
C07810=1082.289,89.294,-65.027,174.438,21.390,153.590
C07811=1082.295,89.544,-65.044,174.440,21.393,153.590
C07812=1082.301,89.793,-65.062,174.442,21.395,153.590
C07813=1082.307,90.042,-65.080,174.444,21.397,153.590
C07814=1082.313,90.292,-65.098,174.445,21.399,153.590
C07815=1082.318,90.541,-65.115,174.448,21.401,153.590
C07816=1082.324,90.791,-65.133,174.449,21.403,153.590
C07817=1082.330,91.039,-65.151,174.451,21.405,153.590
C07818=1082.335,91.289,-65.170,174.453,21.407,153.591
C07819=1082.341,91.538,-65.187,174.455,21.409,153.591
C07820=1082.347,91.787,-65.205,174.456,21.411,153.591
C07821=1082.353,92.037,-65.223,174.457,21.413,153.591
C07822=1082.357,92.286,-65.241,174.460,21.416,153.591
C07823=1082.364,92.536,-65.259,174.461,21.418,153.591
C07824=1082.369,92.784,-65.277,174.463,21.420,153.592
C07825=1082.375,93.033,-65.295,174.465,21.422,153.592
C07826=1082.380,93.284,-65.313,174.467,21.424,153.592
C07827=1082.386,93.533,-65.331,174.468,21.426,153.592
C07828=1082.392,93.782,-65.349,174.470,21.429,153.592
C07829=1082.398,94.031,-65.367,174.472,21.431,153.592
C07830=1082.403,94.280,-65.385,174.474,21.433,153.593
C07831=1082.409,94.530,-65.403,174.475,21.435,153.593
C07832=1082.414,94.779,-65.421,174.478,21.437,153.593
C07833=1082.421,95.059,-65.442,174.480,21.440,153.593
C07834=1082.428,95.338,-65.462,174.481,21.442,153.593
C07835=1082.434,95.617,-65.482,174.483,21.444,153.593
C07836=1082.440,95.897,-65.503,174.485,21.447,153.594
C07837=1082.445,96.146,-65.520,174.487,21.449,153.594
C07838=1082.452,96.395,-65.539,174.489,21.451,153.594
C07839=1082.456,96.644,-65.557,174.490,21.453,153.594
C07840=1082.462,96.894,-65.575,174.493,21.455,153.594
C07841=1082.468,97.142,-65.593,174.494,21.457,153.594
C07842=1082.474,97.393,-65.612,174.496,21.459,153.594
C07843=1082.479,97.642,-65.630,174.498,21.461,153.595
C07844=1082.486,97.891,-65.648,174.500,21.464,153.595
C07845=1082.490,98.140,-65.666,174.501,21.466,153.595
C07846=1082.496,98.390,-65.684,174.503,21.468,153.595
C07847=1082.503,98.639,-65.703,174.505,21.470,153.595
C07848=1082.508,98.888,-65.721,174.507,21.472,153.595
C07849=1082.514,99.137,-65.740,174.508,21.474,153.595
C07850=1082.520,99.386,-65.757,174.511,21.476,153.596
C07851=1082.525,99.637,-65.776,174.512,21.478,153.596
C07852=1082.531,99.885,-65.794,174.514,21.480,153.596
C07853=1082.537,100.135,-65.812,174.516,21.482,153.596
C07854=1082.542,100.383,-65.831,174.518,21.485,153.596
C07855=1082.548,100.633,-65.849,174.519,21.486,153.596
C07856=1082.554,100.882,-65.867,174.522,21.488,153.596
C07857=1082.559,101.132,-65.886,174.523,21.490,153.596
C07858=1082.566,101.381,-65.904,174.525,21.493,153.597
C07859=1082.571,101.630,-65.922,174.526,21.495,153.597
C07860=1082.577,101.879,-65.941,174.529,21.497,153.597
C07861=1082.582,102.129,-65.959,174.531,21.499,153.597
C07862=1082.588,102.378,-65.978,174.532,21.501,153.597
C07863=1082.593,102.627,-65.996,174.535,21.503,153.597
C07864=1082.599,102.876,-66.015,174.536,21.505,153.597
C07865=1082.604,103.125,-66.033,174.538,21.508,153.598
C07866=1082.610,103.375,-66.052,174.540,21.509,153.598
C07867=1082.615,103.624,-66.070,174.542,21.512,153.598
C07868=1082.621,103.873,-66.089,174.543,21.514,153.598
C07869=1082.627,104.123,-66.108,174.545,21.516,153.598
C07870=1082.632,104.372,-66.126,174.547,21.518,153.598
C07871=1082.639,104.621,-66.144,174.549,21.520,153.598
C07872=1082.643,104.870,-66.163,174.551,21.522,153.599
C07873=1082.649,105.120,-66.182,174.553,21.524,153.599
C07874=1082.655,105.368,-66.200,174.554,21.526,153.599
C07875=1082.660,105.618,-66.219,174.556,21.529,153.599
C07876=1082.667,105.867,-66.237,174.558,21.531,153.599
C07877=1082.672,106.116,-66.256,174.560,21.532,153.599
C07878=1082.677,106.366,-66.275,174.561,21.534,153.599
C07879=1082.683,106.615,-66.293,174.564,21.537,153.600
C07880=1082.689,106.864,-66.312,174.566,21.539,153.600
C07881=1082.695,107.114,-66.330,174.567,21.541,153.600
C07882=1082.700,107.362,-66.349,174.570,21.543,153.600
C07883=1082.706,107.612,-66.368,174.571,21.545,153.600
C07884=1082.712,107.861,-66.387,174.573,21.547,153.600
C07885=1082.717,108.110,-66.405,174.575,21.549,153.600
C07886=1082.723,108.360,-66.424,174.577,21.551,153.600
C07887=1082.729,108.609,-66.443,174.578,21.553,153.601
C07888=1082.734,108.858,-66.462,174.581,21.555,153.601
C07889=1082.740,109.107,-66.480,174.582,21.557,153.601
C07890=1082.746,109.357,-66.499,174.584,21.560,153.601
C07891=1082.751,109.606,-66.518,174.586,21.561,153.601
C07892=1082.757,109.855,-66.537,174.588,21.563,153.601
C07893=1082.763,110.105,-66.555,174.590,21.566,153.601
C07894=1082.768,110.353,-66.574,174.592,21.567,153.601
C07895=1082.774,110.603,-66.593,174.594,21.570,153.601
C07896=1082.780,110.852,-66.612,174.595,21.571,153.602
C07897=1082.786,111.131,-66.633,174.598,21.574,153.602
C07898=1082.793,111.411,-66.654,174.600,21.576,153.602
C07899=1082.799,111.690,-66.675,174.602,21.579,153.602
C07900=1082.806,111.970,-66.696,174.604,21.581,153.602
C07901=1082.812,112.219,-66.716,174.606,21.582,153.602
C07902=1082.816,112.469,-66.734,174.608,21.585,153.602
C07903=1082.822,112.718,-66.753,174.609,21.587,153.603
C07904=1082.828,112.967,-66.772,174.612,21.589,153.603
C07905=1082.834,113.216,-66.790,174.613,21.590,153.603
C07906=1082.839,113.465,-66.810,174.615,21.593,153.603
C07907=1082.845,113.715,-66.829,174.618,21.595,153.603
C07908=1082.851,113.964,-66.848,174.619,21.597,153.603
C07909=1082.856,114.213,-66.866,174.621,21.599,153.603
C07910=1082.862,114.462,-66.886,174.623,21.601,153.603
C07911=1082.868,114.711,-66.905,174.625,21.603,153.603
C07912=1082.873,114.960,-66.924,174.627,21.605,153.604
C07913=1082.879,115.210,-66.943,174.629,21.607,153.604
C07914=1082.884,115.459,-66.962,174.631,21.609,153.604
C07915=1082.889,115.708,-66.981,174.632,21.611,153.604
C07916=1082.895,115.957,-67.000,174.635,21.614,153.604
C07917=1082.901,116.207,-67.020,174.636,21.615,153.604
C07918=1082.906,116.456,-67.039,174.638,21.618,153.604
C07919=1082.911,116.705,-67.058,174.641,21.620,153.604
C07920=1082.917,116.954,-67.077,174.642,21.622,153.605
C07921=1082.923,117.204,-67.096,174.644,21.624,153.605
C07922=1082.929,117.453,-67.116,174.646,21.626,153.605
C07923=1082.934,117.702,-67.134,174.648,21.628,153.605
C07924=1082.939,117.951,-67.154,174.649,21.630,153.605
C07925=1082.945,118.201,-67.173,174.652,21.632,153.605
C07926=1082.950,118.449,-67.192,174.654,21.634,153.605
C07927=1082.956,118.698,-67.212,174.655,21.636,153.605
C07928=1082.962,118.948,-67.231,174.658,21.638,153.606
C07929=1082.967,119.197,-67.250,174.659,21.640,153.606
C07930=1082.973,119.447,-67.269,174.661,21.642,153.606
C07931=1082.978,119.695,-67.288,174.664,21.645,153.606
C07932=1082.984,119.945,-67.308,174.665,21.646,153.606
C07933=1082.990,120.194,-67.327,174.667,21.648,153.606
C07934=1082.996,120.443,-67.347,174.669,21.650,153.606
C07935=1083.001,120.692,-67.366,174.671,21.652,153.606
C07936=1083.006,120.941,-67.385,174.673,21.654,153.606
C07937=1083.012,121.191,-67.404,174.675,21.656,153.607
C07938=1083.018,121.440,-67.423,174.677,21.658,153.607
C07939=1083.024,121.689,-67.443,174.679,21.660,153.607
C07940=1083.029,121.938,-67.463,174.681,21.663,153.607
C07941=1083.035,122.187,-67.481,174.683,21.664,153.607
C07942=1083.039,122.437,-67.501,174.685,21.666,153.607
C07943=1083.045,122.685,-67.521,174.687,21.669,153.607
C07944=1083.051,122.935,-67.541,174.688,21.670,153.607
C07945=1083.057,123.184,-67.560,174.691,21.672,153.607
C07946=1083.063,123.434,-67.579,174.693,21.674,153.607
C07947=1083.068,123.682,-67.599,174.694,21.676,153.608
C07948=1083.074,123.931,-67.618,174.697,21.679,153.608
C07949=1083.079,124.181,-67.637,174.698,21.680,153.608
C07950=1083.085,124.430,-67.657,174.700,21.682,153.608
C07951=1083.091,124.679,-67.676,174.703,21.684,153.608
C07952=1083.097,124.928,-67.696,174.704,21.686,153.608
C07953=1083.102,125.178,-67.716,174.706,21.689,153.608
C07954=1083.108,125.427,-67.735,174.709,21.690,153.608
C07955=1083.113,125.676,-67.755,174.710,21.692,153.608
C07956=1083.119,125.925,-67.775,174.713,21.694,153.608
C07957=1083.124,126.174,-67.793,174.714,21.696,153.609
C07958=1083.130,126.423,-67.813,174.716,21.698,153.609
C07959=1083.136,126.672,-67.833,174.719,21.700,153.609
C07960=1083.142,126.922,-67.852,174.720,21.702,153.609
C07961=1083.148,127.201,-67.875,174.722,21.704,153.609
C07962=1083.154,127.481,-67.897,174.725,21.706,153.609
C07963=1083.161,127.761,-67.918,174.727,21.708,153.609
C07964=1083.168,128.040,-67.941,174.729,21.711,153.609
C07965=1083.173,128.289,-67.960,174.732,21.713,153.609
C07966=1083.179,128.537,-67.980,174.733,21.714,153.609
C07967=1083.184,128.787,-67.999,174.735,21.717,153.610
C07968=1083.190,129.036,-68.019,174.738,21.719,153.610
C07969=1083.195,129.285,-68.039,174.739,21.721,153.610
C07970=1083.201,129.534,-68.059,174.742,21.722,153.610
C07971=1083.207,129.784,-68.078,174.744,21.725,153.610
C07972=1083.213,130.032,-68.098,174.745,21.726,153.610
C07973=1083.219,130.282,-68.117,174.748,21.729,153.610
C07974=1083.224,130.531,-68.138,174.749,21.730,153.610
C07975=1083.230,130.780,-68.158,174.752,21.732,153.610
C07976=1083.236,131.029,-68.177,174.754,21.734,153.610
C07977=1083.242,131.278,-68.197,174.755,21.736,153.610
C07978=1083.247,131.528,-68.216,174.758,21.738,153.610
C07979=1083.254,131.777,-68.236,174.760,21.740,153.610
C07980=1083.259,132.026,-68.257,174.761,21.742,153.611
C07981=1083.265,132.276,-68.276,174.764,21.744,153.611
C07982=1083.271,132.524,-68.296,174.766,21.746,153.611
C07983=1083.276,132.774,-68.316,174.768,21.747,153.611
C07984=1083.282,133.023,-68.336,174.770,21.750,153.611
C07985=1083.287,133.272,-68.357,174.772,21.751,153.611
C07986=1083.293,133.522,-68.376,174.774,21.753,153.611
C07987=1083.299,133.770,-68.396,174.776,21.755,153.611
C07988=1083.304,134.019,-68.416,174.778,21.758,153.611
C07989=1083.310,134.269,-68.436,174.780,21.759,153.611
C07990=1083.315,134.518,-68.456,174.782,21.761,153.612
C07991=1083.321,134.767,-68.476,174.785,21.763,153.612
C07992=1083.327,135.016,-68.496,174.786,21.765,153.612
C07993=1083.332,135.265,-68.516,174.788,21.767,153.612
C07994=1083.338,135.514,-68.536,174.791,21.769,153.612
C07995=1083.343,135.763,-68.556,174.792,21.771,153.612
C07996=1083.349,136.012,-68.576,174.795,21.773,153.612
C07997=1083.354,136.262,-68.596,174.797,21.775,153.612
C07998=1083.360,136.511,-68.616,174.799,21.776,153.612
C07999=1083.365,136.760,-68.637,174.801,21.779,153.612
C08000=1083.371,137.009,-68.657,174.803,21.781,153.612
C08001=1083.376,137.258,-68.677,174.805,21.782,153.612
C08002=1083.382,137.507,-68.696,174.807,21.784,153.612
C08003=1083.388,137.756,-68.716,174.809,21.787,153.613
C08004=1083.393,138.005,-68.737,174.811,21.788,153.613
C08005=1083.399,138.254,-68.757,174.813,21.790,153.613
C08006=1083.405,138.503,-68.778,174.815,21.792,153.613
C08007=1083.411,138.753,-68.798,174.817,21.794,153.613
C08008=1083.416,139.002,-68.818,174.819,21.796,153.613
C08009=1083.421,139.251,-68.838,174.822,21.798,153.613
C08010=1083.427,139.500,-68.858,174.824,21.800,153.613
C08011=1083.433,139.749,-68.879,174.826,21.802,153.613
C08012=1083.439,139.998,-68.899,174.828,21.803,153.613
C08013=1083.444,140.247,-68.919,174.830,21.806,153.613
C08014=1083.450,140.496,-68.939,174.832,21.807,153.613
C08015=1083.455,140.745,-68.960,174.834,21.810,153.614
C08016=1083.461,140.995,-68.981,174.836,21.811,153.614
C08017=1083.467,141.244,-69.001,174.838,21.813,153.614
C08018=1083.472,141.493,-69.021,174.840,21.815,153.614
C08019=1083.478,141.742,-69.041,174.843,21.817,153.614
C08020=1083.484,141.991,-69.062,174.845,21.819,153.614
C08021=1083.489,142.240,-69.082,174.846,21.821,153.614
C08022=1083.495,142.489,-69.102,174.849,21.823,153.614
C08023=1083.500,142.738,-69.123,174.851,21.825,153.614
C08024=1083.505,142.987,-69.143,174.853,21.826,153.614
C08025=1083.512,143.266,-69.166,174.855,21.829,153.614
C08026=1083.519,143.546,-69.189,174.857,21.831,153.614
C08027=1083.525,143.826,-69.212,174.861,21.833,153.614
C08028=1083.531,144.105,-69.235,174.863,21.835,153.614
C08029=1083.537,144.354,-69.255,174.864,21.837,153.615
C08030=1083.542,144.603,-69.276,174.867,21.839,153.615
C08031=1083.547,144.852,-69.296,174.869,21.841,153.615
C08032=1083.553,145.102,-69.317,174.871,21.843,153.615
C08033=1083.559,145.350,-69.337,174.873,21.845,153.615
C08034=1083.565,145.600,-69.359,174.875,21.847,153.615
C08035=1083.570,145.849,-69.379,174.878,21.849,153.615
C08036=1083.576,146.098,-69.399,174.879,21.850,153.615
C08037=1083.581,146.347,-69.420,174.882,21.853,153.615
C08038=1083.587,146.597,-69.441,174.884,21.854,153.615
C08039=1083.592,146.846,-69.461,174.886,21.856,153.615
C08040=1083.599,147.094,-69.482,174.888,21.858,153.615
C08041=1083.604,147.343,-69.502,174.890,21.860,153.615
C08042=1083.609,147.592,-69.523,174.893,21.862,153.615
C08043=1083.615,147.842,-69.544,174.895,21.864,153.615
C08044=1083.621,148.091,-69.564,174.896,21.866,153.616
C08045=1083.627,148.339,-69.585,174.899,21.867,153.616
C08046=1083.632,148.588,-69.606,174.901,21.869,153.616
C08047=1083.638,148.838,-69.627,174.903,21.871,153.616
C08048=1083.643,149.087,-69.648,174.905,21.873,153.616
C08049=1083.649,149.336,-69.668,174.908,21.875,153.616
C08050=1083.655,149.585,-69.688,174.910,21.877,153.616
C08051=1083.660,149.834,-69.709,174.911,21.879,153.616
C08052=1083.666,150.083,-69.731,174.914,21.880,153.616
C08053=1083.671,150.332,-69.751,174.916,21.883,153.616
C08054=1083.676,150.581,-69.772,174.919,21.885,153.616
C08055=1083.683,150.830,-69.793,174.921,21.886,153.616
C08056=1083.688,151.080,-69.814,174.922,21.888,153.616
C08057=1083.693,151.329,-69.834,174.925,21.890,153.616
C08058=1083.699,151.577,-69.856,174.927,21.892,153.616
C08059=1083.705,151.827,-69.877,174.930,21.894,153.616
C08060=1083.710,152.075,-69.898,174.931,21.896,153.616
C08061=1083.716,152.324,-69.918,174.934,21.898,153.616
C08062=1083.722,152.574,-69.939,174.936,21.900,153.616
C08063=1083.728,152.823,-69.960,174.938,21.902,153.617
C08064=1083.733,153.072,-69.981,174.940,21.903,153.617
C08065=1083.738,153.304,-70.001,174.942,21.905,153.617
C08066=1083.743,153.538,-70.020,174.945,21.907,153.617
C08067=1083.748,153.772,-70.040,174.946,21.908,153.617
C08068=1083.754,154.004,-70.060,174.948,21.911,153.617
C08069=1083.759,154.237,-70.079,174.950,21.912,153.617
C08070=1083.764,154.470,-70.099,174.952,21.914,153.617
C08071=1083.770,154.704,-70.118,174.955,21.916,153.617
C08072=1083.775,154.936,-70.138,174.957,21.917,153.617
C08073=1083.780,155.185,-70.159,174.959,21.920,153.617
C08074=1083.786,155.434,-70.180,174.961,21.921,153.617
C08075=1083.792,155.683,-70.201,174.964,21.923,153.617
C08076=1083.797,155.932,-70.223,174.965,21.925,153.617
C08077=1083.803,156.182,-70.244,174.967,21.927,153.617
C08078=1083.808,156.431,-70.265,174.970,21.929,153.617
C08079=1083.814,156.679,-70.286,174.972,21.931,153.617
C08080=1083.819,156.929,-70.307,174.975,21.932,153.617
C08081=1083.825,157.177,-70.328,174.976,21.934,153.618
C08082=1083.830,157.426,-70.349,174.979,21.936,153.618
C08083=1083.836,157.676,-70.371,174.981,21.938,153.618
C08084=1083.842,157.924,-70.392,174.984,21.940,153.618
C08085=1083.847,158.173,-70.412,174.986,21.942,153.618
C08086=1083.853,158.423,-70.435,174.987,21.944,153.618
C08087=1083.858,158.672,-70.455,174.990,21.945,153.618
C08088=1083.864,158.921,-70.477,174.992,21.947,153.618
C08089=1083.871,159.232,-70.503,174.994,21.950,153.618
C08090=1083.878,159.543,-70.530,174.998,21.952,153.618
C08091=1083.885,159.854,-70.557,175.000,21.954,153.618
C08092=1083.892,160.165,-70.583,175.003,21.957,153.618
C08093=1083.898,160.415,-70.605,175.006,21.958,153.618
C08094=1083.903,160.664,-70.626,175.008,21.960,153.618
C08095=1083.909,160.913,-70.647,175.010,21.962,153.618
C08096=1083.915,161.161,-70.668,175.012,21.964,153.618
C08097=1083.921,161.411,-70.690,175.015,21.966,153.618
C08098=1083.925,161.660,-70.711,175.017,21.968,153.618
C08099=1083.931,161.908,-70.733,175.019,21.969,153.618
C08100=1083.937,162.158,-70.754,175.022,21.972,153.618
C08101=1083.942,162.407,-70.776,175.023,21.973,153.619
C08102=1083.947,162.656,-70.797,175.026,21.975,153.619
C08103=1083.953,162.905,-70.819,175.028,21.977,153.619
C08104=1083.958,163.154,-70.840,175.030,21.979,153.619
C08105=1083.964,163.403,-70.862,175.033,21.981,153.619
C08106=1083.969,163.652,-70.884,175.035,21.983,153.619
C08107=1083.975,163.900,-70.905,175.037,21.985,153.619
C08108=1083.980,164.150,-70.927,175.039,21.987,153.619
C08109=1083.985,164.399,-70.948,175.042,21.988,153.619
C08110=1083.991,164.648,-70.970,175.044,21.991,153.619
C08111=1083.996,164.897,-70.991,175.046,21.993,153.619
C08112=1084.001,165.146,-71.013,175.049,21.994,153.619
C08113=1084.007,165.395,-71.035,175.050,21.996,153.619
C08114=1084.012,165.644,-71.056,175.053,21.998,153.619
C08115=1084.018,165.893,-71.078,175.055,22.000,153.619
C08116=1084.023,166.142,-71.100,175.057,22.002,153.619
C08117=1084.029,166.391,-71.122,175.060,22.004,153.619
C08118=1084.035,166.639,-71.143,175.062,22.006,153.619
C08119=1084.040,166.889,-71.165,175.065,22.008,153.620
C08120=1084.046,167.137,-71.186,175.066,22.009,153.620
C08121=1084.051,167.387,-71.209,175.069,22.011,153.620
C08122=1084.057,167.635,-71.230,175.071,22.013,153.620
C08123=1084.062,167.885,-71.252,175.073,22.015,153.620
C08124=1084.068,168.133,-71.273,175.076,22.017,153.620
C08125=1084.073,168.383,-71.296,175.078,22.019,153.620
C08126=1084.078,168.632,-71.317,175.081,22.021,153.620
C08127=1084.084,168.881,-71.339,175.083,22.023,153.620
C08128=1084.089,169.130,-71.361,175.084,22.025,153.620
C08129=1084.095,169.379,-71.383,175.087,22.026,153.620
C08130=1084.100,169.628,-71.404,175.089,22.028,153.620
C08131=1084.106,169.877,-71.426,175.092,22.030,153.620
C08132=1084.111,170.125,-71.449,175.094,22.032,153.620
C08133=1084.117,170.374,-71.470,175.097,22.034,153.620
C08134=1084.122,170.623,-71.492,175.099,22.036,153.620
C08135=1084.128,170.872,-71.514,175.101,22.038,153.620
C08136=1084.133,171.121,-71.536,175.103,22.039,153.620
C08137=1084.139,171.371,-71.557,175.105,22.041,153.620
C08138=1084.145,171.619,-71.580,175.108,22.043,153.620
C08139=1084.150,171.868,-71.602,175.110,22.045,153.620
C08140=1084.156,172.117,-71.624,175.113,22.047,153.620
C08141=1084.161,172.366,-71.646,175.115,22.048,153.620
C08142=1084.167,172.615,-71.667,175.118,22.051,153.620
C08143=1084.173,172.864,-71.690,175.120,22.053,153.620
C08144=1084.178,173.113,-71.711,175.122,22.054,153.620
C08145=1084.184,173.362,-71.734,175.125,22.056,153.620
C08146=1084.189,173.611,-71.756,175.126,22.058,153.621
C08147=1084.195,173.860,-71.778,175.129,22.059,153.621
C08148=1084.201,174.109,-71.800,175.131,22.061,153.621
C08149=1084.206,174.358,-71.821,175.134,22.063,153.621
C08150=1084.212,174.607,-71.844,175.136,22.065,153.621
C08151=1084.217,174.856,-71.867,175.139,22.067,153.621
C08152=1084.223,175.105,-71.888,175.141,22.069,153.621
C08153=1084.230,175.384,-71.913,175.143,22.071,153.621
C08154=1084.235,175.662,-71.938,175.146,22.073,153.621
C08155=1084.241,175.941,-71.963,175.149,22.075,153.621
C08156=1084.248,176.221,-71.988,175.152,22.077,153.621
C08157=1084.254,176.468,-72.010,175.154,22.079,153.621
C08158=1084.259,176.718,-72.032,175.157,22.081,153.621
C08159=1084.265,176.967,-72.054,175.159,22.082,153.621
C08160=1084.271,177.215,-72.076,175.161,22.084,153.621
C08161=1084.276,177.465,-72.098,175.164,22.086,153.621
C08162=1084.282,177.714,-72.121,175.166,22.088,153.621
C08163=1084.288,177.963,-72.143,175.169,22.090,153.621
C08164=1084.293,178.211,-72.166,175.170,22.091,153.621
C08165=1084.299,178.461,-72.188,175.173,22.093,153.621
C08166=1084.305,178.709,-72.210,175.175,22.095,153.621
C08167=1084.311,178.959,-72.232,175.178,22.097,153.621
C08168=1084.316,179.207,-72.255,175.180,22.098,153.621
C08169=1084.322,179.456,-72.277,175.183,22.100,153.621
C08170=1084.328,179.705,-72.299,175.185,22.102,153.621
C08171=1084.333,179.955,-72.322,175.188,22.104,153.621
C08172=1084.338,180.203,-72.344,175.190,22.106,153.621
C08173=1084.344,180.452,-72.366,175.192,22.108,153.621
C08174=1084.350,180.701,-72.389,175.195,22.109,153.621
C08175=1084.355,180.950,-72.411,175.197,22.111,153.621
C08176=1084.362,181.199,-72.433,175.200,22.113,153.621
C08177=1084.367,181.447,-72.456,175.202,22.115,153.621
C08178=1084.372,181.697,-72.478,175.205,22.117,153.621
C08179=1084.378,181.946,-72.501,175.207,22.119,153.621
C08180=1084.384,182.195,-72.523,175.210,22.120,153.621
C08181=1084.390,182.444,-72.546,175.212,22.122,153.621
C08182=1084.396,182.693,-72.569,175.215,22.123,153.621
C08183=1084.401,182.941,-72.591,175.217,22.125,153.621
C08184=1084.407,183.190,-72.613,175.220,22.127,153.621
C08185=1084.413,183.439,-72.636,175.222,22.129,153.621
C08186=1084.418,183.688,-72.658,175.224,22.130,153.621
C08187=1084.424,183.937,-72.681,175.226,22.132,153.621
C08188=1084.430,184.186,-72.703,175.229,22.134,153.621
C08189=1084.436,184.435,-72.726,175.231,22.136,153.621
C08190=1084.441,184.684,-72.748,175.233,22.138,153.621
C08191=1084.447,184.933,-72.771,175.236,22.139,153.621
C08192=1084.452,185.181,-72.794,175.239,22.141,153.621
C08193=1084.458,185.430,-72.817,175.241,22.143,153.621
C08194=1084.464,185.680,-72.839,175.243,22.145,153.621
C08195=1084.469,185.928,-72.862,175.246,22.147,153.621
C08196=1084.474,186.177,-72.885,175.248,22.149,153.621
C08197=1084.480,186.426,-72.908,175.251,22.150,153.621
C08198=1084.486,186.675,-72.931,175.253,22.152,153.621
C08199=1084.491,186.924,-72.953,175.256,22.154,153.621
C08200=1084.496,187.173,-72.976,175.258,22.156,153.621
C08201=1084.502,187.422,-72.999,175.260,22.158,153.621
C08202=1084.507,187.671,-73.022,175.263,22.160,153.622
C08203=1084.513,187.919,-73.045,175.265,22.162,153.622
C08204=1084.519,188.168,-73.068,175.268,22.164,153.622
C08205=1084.524,188.417,-73.090,175.270,22.166,153.622
C08206=1084.529,188.666,-73.114,175.273,22.167,153.622
C08207=1084.535,188.915,-73.137,175.275,22.169,153.622
C08208=1084.540,189.164,-73.159,175.277,22.171,153.622
C08209=1084.546,189.413,-73.182,175.280,22.173,153.622
C08210=1084.551,189.662,-73.205,175.283,22.175,153.622
C08211=1084.557,189.911,-73.228,175.286,22.177,153.622
C08212=1084.562,190.159,-73.251,175.288,22.179,153.622
C08213=1084.567,190.408,-73.274,175.291,22.181,153.622
C08214=1084.573,190.657,-73.297,175.293,22.182,153.622
C08215=1084.579,190.906,-73.320,175.296,22.184,153.622
C08216=1084.584,191.155,-73.343,175.298,22.186,153.622
C08217=1084.590,191.433,-73.369,175.300,22.188,153.622
C08218=1084.597,191.712,-73.396,175.303,22.190,153.622
C08219=1084.603,191.990,-73.420,175.306,22.193,153.622
C08220=1084.609,192.268,-73.447,175.309,22.194,153.622
C08221=1084.615,192.517,-73.469,175.311,22.196,153.622
C08222=1084.620,192.766,-73.493,175.313,22.198,153.622
C08223=1084.625,193.015,-73.516,175.316,22.200,153.622
C08224=1084.631,193.264,-73.539,175.318,22.202,153.622
C08225=1084.637,193.513,-73.562,175.322,22.204,153.622
C08226=1084.642,193.762,-73.586,175.324,22.206,153.622
C08227=1084.648,194.011,-73.609,175.327,22.208,153.622
C08228=1084.654,194.259,-73.632,175.329,22.209,153.622
C08229=1084.659,194.508,-73.655,175.332,22.211,153.622
C08230=1084.664,194.758,-73.678,175.334,22.213,153.622
C08231=1084.670,195.006,-73.701,175.336,22.215,153.622
C08232=1084.676,195.255,-73.725,175.339,22.217,153.622
C08233=1084.682,195.504,-73.748,175.341,22.218,153.622
C08234=1084.687,195.753,-73.772,175.344,22.220,153.622
C08235=1084.693,196.002,-73.795,175.346,22.222,153.622
C08236=1084.699,196.250,-73.818,175.349,22.223,153.622
C08237=1084.704,196.499,-73.842,175.351,22.225,153.622
C08238=1084.709,196.748,-73.865,175.354,22.227,153.622
C08239=1084.715,196.997,-73.888,175.356,22.229,153.622
C08240=1084.720,197.246,-73.912,175.360,22.231,153.622
C08241=1084.726,197.494,-73.935,175.362,22.233,153.622
C08242=1084.732,197.743,-73.958,175.365,22.235,153.622
C08243=1084.738,197.992,-73.981,175.367,22.237,153.622
C08244=1084.743,198.241,-74.005,175.369,22.238,153.622
C08245=1084.749,198.490,-74.028,175.372,22.240,153.622
C08246=1084.755,198.739,-74.052,175.374,22.242,153.622
C08247=1084.760,198.988,-74.075,175.377,22.244,153.622
C08248=1084.766,199.237,-74.098,175.379,22.246,153.622
C08249=1084.772,199.485,-74.122,175.382,22.247,153.622
C08250=1084.777,199.734,-74.146,175.384,22.249,153.622
C08251=1084.783,199.983,-74.169,175.388,22.251,153.622
C08252=1084.788,200.232,-74.193,175.390,22.253,153.622
C08253=1084.794,200.481,-74.216,175.393,22.255,153.622
C08254=1084.800,200.730,-74.240,175.395,22.257,153.622
C08255=1084.805,200.979,-74.263,175.398,22.258,153.622
C08256=1084.811,201.227,-74.287,175.400,22.260,153.622
C08257=1084.817,201.476,-74.310,175.403,22.262,153.622
C08258=1084.822,201.725,-74.334,175.405,22.263,153.622
C08259=1084.828,201.974,-74.357,175.408,22.265,153.622
C08260=1084.833,202.222,-74.381,175.411,22.267,153.622
C08261=1084.840,202.472,-74.405,175.413,22.269,153.622
C08262=1084.846,202.720,-74.428,175.416,22.271,153.622
C08263=1084.851,202.969,-74.452,175.418,22.273,153.622
C08264=1084.856,203.218,-74.476,175.421,22.275,153.622
C08265=1084.862,203.466,-74.500,175.423,22.277,153.622
C08266=1084.867,203.715,-74.523,175.426,22.278,153.622
C08267=1084.873,203.964,-74.547,175.428,22.280,153.622
C08268=1084.878,204.213,-74.571,175.432,22.283,153.622
C08269=1084.884,204.462,-74.595,175.434,22.284,153.622
C08270=1084.890,204.710,-74.619,175.436,22.286,153.622
C08271=1084.895,204.960,-74.642,175.439,22.288,153.622
C08272=1084.901,205.208,-74.666,175.441,22.290,153.622
C08273=1084.906,205.456,-74.690,175.444,22.292,153.622
C08274=1084.911,205.706,-74.714,175.447,22.294,153.622
C08275=1084.918,205.955,-74.738,175.450,22.296,153.622
C08276=1084.923,206.203,-74.762,175.452,22.298,153.622
C08277=1084.928,206.452,-74.786,175.455,22.299,153.622
C08278=1084.934,206.701,-74.809,175.457,22.301,153.622
C08279=1084.940,206.949,-74.834,175.459,22.303,153.623
C08280=1084.946,207.199,-74.858,175.462,22.305,153.623
C08281=1084.969,208.227,-74.956,175.546,22.349,153.619
C08282=1084.978,208.616,-74.995,175.551,22.354,153.620
C08283=1084.987,209.005,-75.033,175.554,22.358,153.620
C08284=1084.995,209.395,-75.071,175.558,22.362,153.621
C08285=1085.004,209.785,-75.110,175.562,22.366,153.621
C08286=1085.009,210.033,-75.134,175.565,22.369,153.621
C08287=1085.015,210.281,-75.159,175.567,22.372,153.621
C08288=1085.021,210.531,-75.184,175.570,22.375,153.622
C08289=1085.026,210.779,-75.208,175.572,22.377,153.622
C08290=1085.032,211.029,-75.232,175.574,22.380,153.622
C08291=1085.037,211.277,-75.257,175.577,22.383,153.622
C08292=1085.044,211.526,-75.282,175.579,22.386,153.622
C08293=1085.049,211.774,-75.306,175.581,22.389,153.623
C08294=1085.054,212.023,-75.330,175.585,22.391,153.623
C08295=1085.060,212.272,-75.356,175.587,22.394,153.623
C08296=1085.066,212.520,-75.380,175.590,22.397,153.623
C08297=1085.072,212.770,-75.405,175.592,22.400,153.624
C08298=1085.077,213.018,-75.429,175.594,22.402,153.624
C08299=1085.083,213.267,-75.454,175.597,22.405,153.624
C08300=1085.088,213.515,-75.479,175.599,22.408,153.624
C08301=1085.094,213.765,-75.503,175.602,22.411,153.625
C08302=1085.100,214.013,-75.528,175.605,22.414,153.625
C08303=1085.106,214.262,-75.553,175.607,22.416,153.625
C08304=1085.111,214.510,-75.578,175.610,22.420,153.625
C08305=1085.116,214.759,-75.603,175.612,22.422,153.625
C08306=1085.122,215.008,-75.627,175.615,22.425,153.626
C08307=1085.127,215.256,-75.652,175.617,22.428,153.626
C08308=1085.133,215.505,-75.677,175.620,22.431,153.626
C08309=1085.139,215.753,-75.702,175.622,22.434,153.626
C08310=1085.145,216.003,-75.726,175.625,22.436,153.627
C08311=1085.150,216.252,-75.752,175.627,22.439,153.627
C08312=1085.156,216.500,-75.777,175.630,22.442,153.627
C08313=1085.162,216.749,-75.802,175.633,22.445,153.627
C08314=1085.167,216.997,-75.826,175.635,22.448,153.627
C08315=1085.173,217.246,-75.852,175.637,22.450,153.628
C08316=1085.178,217.495,-75.876,175.640,22.453,153.628
C08317=1085.184,217.744,-75.902,175.642,22.456,153.628
C08318=1085.189,217.992,-75.926,175.645,22.459,153.628
C08319=1085.196,218.241,-75.951,175.647,22.462,153.629
C08320=1085.200,218.489,-75.977,175.650,22.465,153.629
C08321=1085.206,218.738,-76.002,175.653,22.467,153.629
C08322=1085.213,218.987,-76.027,175.655,22.470,153.629
C08323=1085.218,219.236,-76.051,175.658,22.473,153.629
C08324=1085.223,219.485,-76.077,175.660,22.475,153.630
C08325=1085.229,219.733,-76.102,175.663,22.479,153.630
C08326=1085.235,219.982,-76.127,175.665,22.481,153.630
C08327=1085.241,220.231,-76.152,175.668,22.484,153.630
C08328=1085.246,220.479,-76.178,175.671,22.487,153.631
C08329=1085.252,220.728,-76.202,175.674,22.490,153.631
C08330=1085.258,220.977,-76.227,175.676,22.493,153.631
C08331=1085.264,221.225,-76.252,175.678,22.495,153.631
C08332=1085.269,221.474,-76.278,175.681,22.498,153.632
C08333=1085.275,221.723,-76.303,175.683,22.501,153.632
C08334=1085.284,222.116,-76.343,175.688,22.505,153.632
C08335=1085.292,222.509,-76.383,175.691,22.510,153.633
C08336=1085.301,222.902,-76.423,175.696,22.514,153.633
C08337=1085.310,223.295,-76.464,175.700,22.519,153.633
C08338=1085.316,223.545,-76.488,175.702,22.522,153.634
C08339=1085.321,223.794,-76.514,175.705,22.524,153.634
C08340=1085.327,224.042,-76.539,175.708,22.527,153.634
C08341=1085.332,224.291,-76.565,175.710,22.530,153.634
C08342=1085.339,224.539,-76.590,175.713,22.533,153.634
C08343=1085.344,224.788,-76.616,175.715,22.536,153.635
C08344=1085.350,225.036,-76.641,175.718,22.539,153.635
C08345=1085.355,225.285,-76.667,175.720,22.541,153.635
C08346=1085.361,225.533,-76.692,175.723,22.544,153.635
C08347=1085.366,225.782,-76.718,175.725,22.547,153.636
C08348=1085.372,226.031,-76.743,175.728,22.550,153.636
C08349=1085.378,226.280,-76.769,175.731,22.553,153.636
C08350=1085.384,226.528,-76.794,175.733,22.556,153.636
C08351=1085.389,226.777,-76.820,175.736,22.559,153.637
C08352=1085.394,227.026,-76.846,175.738,22.561,153.637
C08353=1085.400,227.274,-76.871,175.741,22.564,153.637
C08354=1085.406,227.523,-76.897,175.743,22.567,153.637
C08355=1085.412,227.771,-76.922,175.746,22.570,153.637
C08356=1085.417,228.020,-76.948,175.749,22.572,153.638
C08357=1085.423,228.269,-76.974,175.752,22.576,153.638
C08358=1085.428,228.517,-76.999,175.754,22.578,153.638
C08359=1085.435,228.766,-77.025,175.757,22.581,153.638
C08360=1085.440,229.015,-77.051,175.759,22.584,153.639
C08361=1085.445,229.264,-77.076,175.762,22.587,153.639
C08362=1085.452,229.513,-77.102,175.764,22.590,153.639
C08363=1085.457,229.760,-77.128,175.767,22.593,153.639
C08364=1085.463,230.009,-77.153,175.770,22.595,153.639
C08365=1085.469,230.258,-77.179,175.773,22.598,153.640
C08366=1085.474,230.507,-77.205,175.775,22.601,153.640
C08367=1085.480,230.756,-77.231,175.778,22.604,153.640
C08368=1085.485,231.003,-77.257,175.780,22.607,153.640
C08369=1085.491,231.252,-77.283,175.783,22.609,153.641
C08370=1085.496,231.501,-77.309,175.785,22.612,153.641
C08371=1085.502,231.750,-77.334,175.788,22.615,153.641
C08372=1085.508,231.998,-77.361,175.791,22.618,153.641
C08373=1085.514,232.247,-77.387,175.794,22.621,153.642
C08374=1085.519,232.496,-77.412,175.796,22.624,153.642
C08375=1085.525,232.744,-77.438,175.799,22.627,153.642
C08376=1085.531,232.993,-77.464,175.802,22.630,153.642
C08377=1085.536,233.242,-77.490,175.804,22.633,153.643
C08378=1085.542,233.490,-77.517,175.807,22.635,153.643
C08379=1085.547,233.739,-77.543,175.809,22.638,153.643
C08380=1085.554,233.988,-77.568,175.812,22.641,153.643
C08381=1085.559,234.235,-77.594,175.814,22.644,153.644
C08382=1085.564,234.484,-77.620,175.817,22.647,153.644
C08383=1085.570,234.733,-77.646,175.820,22.650,153.644
C08384=1085.575,234.982,-77.673,175.823,22.653,153.644
C08385=1085.581,235.230,-77.699,175.825,22.655,153.644
C08386=1085.589,235.609,-77.739,175.829,22.660,153.645
C08387=1085.598,235.988,-77.779,175.833,22.664,153.645
C08388=1085.607,236.366,-77.819,175.838,22.669,153.646
C08389=1085.615,236.745,-77.858,175.841,22.673,153.646
C08390=1085.621,236.994,-77.885,175.843,22.676,153.646
C08391=1085.626,237.242,-77.912,175.847,22.679,153.646
C08392=1085.632,237.491,-77.937,175.850,22.682,153.647
C08393=1085.638,237.739,-77.964,175.852,22.685,153.647
C08394=1085.643,237.988,-77.990,175.855,22.687,153.647
C08395=1085.649,238.237,-78.017,175.857,22.690,153.647
C08396=1085.654,238.486,-78.043,175.860,22.693,153.648
C08397=1085.661,238.734,-78.069,175.862,22.696,153.648
C08398=1085.667,238.982,-78.095,175.865,22.699,153.648
C08399=1085.672,239.231,-78.121,175.868,22.702,153.648
C08400=1085.678,239.479,-78.148,175.871,22.705,153.649
C08401=1085.684,239.728,-78.175,175.874,22.708,153.649
C08402=1085.689,239.977,-78.201,175.876,22.711,153.649
C08403=1085.695,240.225,-78.227,175.879,22.713,153.649
C08404=1085.701,240.473,-78.254,175.881,22.716,153.650
C08405=1085.706,240.722,-78.281,175.884,22.719,153.650
C08406=1085.711,240.971,-78.307,175.887,22.722,153.650
C08407=1085.717,241.219,-78.334,175.889,22.725,153.650
C08408=1085.723,241.468,-78.360,175.892,22.728,153.650
C08409=1085.728,241.716,-78.387,175.895,22.730,153.651
C08410=1085.734,241.965,-78.413,175.898,22.734,153.651
C08411=1085.740,242.214,-78.440,175.900,22.736,153.651
C08412=1085.746,242.462,-78.466,175.903,22.739,153.651
C08413=1085.751,242.710,-78.493,175.906,22.742,153.652
C08414=1085.757,242.965,-78.520,175.908,22.745,153.652
C08415=1085.763,243.220,-78.548,175.911,22.748,153.652
C08416=1085.769,243.474,-78.575,175.914,22.751,153.652
C08417=1085.775,243.729,-78.602,175.916,22.754,153.653
C08418=1085.780,243.978,-78.629,175.919,22.757,153.653
C08419=1085.786,244.226,-78.656,175.922,22.760,153.653
C08420=1085.791,244.474,-78.682,175.924,22.763,153.653
C08421=1085.797,244.723,-78.709,175.928,22.766,153.654
C08422=1085.802,244.971,-78.736,175.930,22.769,153.654
C08423=1085.808,245.220,-78.763,175.933,22.772,153.654
C08424=1085.814,245.468,-78.789,175.936,22.775,153.654
C08425=1085.820,245.716,-78.816,175.938,22.777,153.655
C08426=1085.825,245.965,-78.843,175.941,22.781,153.655
C08427=1085.831,246.214,-78.870,175.943,22.783,153.655
C08428=1085.837,246.462,-78.897,175.946,22.787,153.655
C08429=1085.842,246.711,-78.924,175.949,22.789,153.656
C08430=1085.848,246.959,-78.951,175.951,22.792,153.656
C08431=1085.853,247.208,-78.978,175.954,22.795,153.656
C08432=1085.858,247.457,-79.005,175.957,22.798,153.656
C08433=1085.864,247.705,-79.031,175.960,22.801,153.657
C08434=1085.870,247.953,-79.058,175.963,22.804,153.657
C08435=1085.875,248.202,-79.085,175.965,22.807,153.657
C08436=1085.882,248.450,-79.113,175.968,22.810,153.657
C08437=1085.887,248.699,-79.140,175.971,22.813,153.658
C08438=1085.895,249.077,-79.181,175.975,22.817,153.658
C08439=1085.904,249.454,-79.223,175.979,22.822,153.659
C08440=1085.912,249.832,-79.264,175.983,22.827,153.659
C08441=1085.920,250.210,-79.305,175.987,22.831,153.659
C08442=1085.926,250.459,-79.332,175.990,22.834,153.660
C08443=1085.932,250.708,-79.359,175.993,22.837,153.660
C08444=1085.937,250.956,-79.386,175.996,22.840,153.660
C08445=1085.943,251.204,-79.414,175.998,22.843,153.660
C08446=1085.948,251.453,-79.441,176.001,22.846,153.661
C08447=1085.954,251.702,-79.468,176.004,22.849,153.661
C08448=1085.960,251.950,-79.496,176.006,22.852,153.661
C08449=1085.965,252.199,-79.523,176.009,22.855,153.661
C08450=1085.970,252.447,-79.550,176.011,22.858,153.662
C08451=1085.976,252.695,-79.578,176.014,22.861,153.662
C08452=1085.982,252.944,-79.605,176.017,22.864,153.662
C08453=1085.988,253.192,-79.633,176.020,22.866,153.662
C08454=1085.993,253.440,-79.659,176.023,22.870,153.663
C08455=1085.998,253.689,-79.687,176.026,22.873,153.663
C08456=1086.005,253.938,-79.714,176.028,22.876,153.663
C08457=1086.010,254.186,-79.742,176.031,22.879,153.664
C08458=1086.015,254.434,-79.770,176.034,22.882,153.664
C08459=1086.021,254.683,-79.796,176.036,22.884,153.664
C08460=1086.027,254.931,-79.825,176.039,22.888,153.664
C08461=1086.033,255.180,-79.851,176.042,22.891,153.665
C08462=1086.038,255.428,-79.879,176.044,22.894,153.665
C08463=1086.044,255.677,-79.907,176.047,22.897,153.665
C08464=1086.050,255.925,-79.934,176.050,22.900,153.665
C08465=1086.055,256.174,-79.961,176.053,22.902,153.666
C08466=1086.062,256.422,-79.989,176.056,22.905,153.666
C08467=1086.067,256.671,-80.016,176.059,22.909,153.666
C08468=1086.072,256.919,-80.044,176.062,22.912,153.666
C08469=1086.079,257.167,-80.072,176.064,22.915,153.667
C08470=1086.084,257.416,-80.099,176.067,22.917,153.667
C08471=1086.089,257.664,-80.127,176.070,22.921,153.667
C08472=1086.096,257.912,-80.155,176.072,22.923,153.667
C08473=1086.101,258.161,-80.182,176.075,22.927,153.668
C08474=1086.106,258.409,-80.210,176.078,22.930,153.668
C08475=1086.113,258.658,-80.238,176.080,22.932,153.668
C08476=1086.118,258.906,-80.265,176.083,22.935,153.668
C08477=1086.124,259.155,-80.293,176.086,22.938,153.669
C08478=1086.130,259.403,-80.321,176.089,22.941,153.669
C08479=1086.135,259.651,-80.349,176.092,22.944,153.669
C08480=1086.141,259.900,-80.376,176.095,22.947,153.669
C08481=1086.147,260.148,-80.404,176.098,22.950,153.670
C08482=1086.153,260.397,-80.432,176.100,22.953,153.670
C08483=1086.158,260.645,-80.460,176.103,22.956,153.670
C08484=1086.165,260.893,-80.488,176.106,22.960,153.670
C08485=1086.170,261.142,-80.515,176.108,22.962,153.671
C08486=1086.175,261.390,-80.543,176.111,22.965,153.671
C08487=1086.181,261.639,-80.571,176.114,22.968,153.671
C08488=1086.187,261.886,-80.599,176.116,22.971,153.671
C08489=1086.193,262.135,-80.627,176.120,22.974,153.672
C08490=1086.202,262.511,-80.669,176.124,22.979,153.672
C08491=1086.211,262.885,-80.711,176.128,22.983,153.672
C08492=1086.219,263.261,-80.753,176.133,22.987,153.673
C08493=1086.229,263.636,-80.796,176.137,22.992,153.673
C08494=1086.234,263.884,-80.824,176.139,22.995,153.673
C08495=1086.240,264.132,-80.852,176.142,22.998,153.674
C08496=1086.245,264.380,-80.880,176.145,23.001,153.674
C08497=1086.251,264.629,-80.908,176.148,23.004,153.674
C08498=1086.257,264.877,-80.936,176.150,23.007,153.675
C08499=1086.262,265.126,-80.965,176.154,23.010,153.675
C08500=1086.268,265.374,-80.992,176.157,23.013,153.675
C08501=1086.274,265.623,-81.021,176.160,23.017,153.675
C08502=1086.279,265.871,-81.049,176.162,23.019,153.676
C08503=1086.285,266.119,-81.078,176.165,23.022,153.676
C08504=1086.291,266.367,-81.106,176.168,23.025,153.676
C08505=1086.297,266.616,-81.134,176.170,23.028,153.676
C08506=1086.302,266.864,-81.162,176.173,23.031,153.677
C08507=1086.308,267.113,-81.190,176.176,23.034,153.677
C08508=1086.313,267.361,-81.218,176.179,23.038,153.677
C08509=1086.319,267.609,-81.247,176.181,23.040,153.678
C08510=1086.325,267.857,-81.275,176.184,23.044,153.678
C08511=1086.331,268.106,-81.304,176.187,23.047,153.678
C08512=1086.337,268.354,-81.332,176.190,23.050,153.678
C08513=1086.342,268.602,-81.360,176.193,23.053,153.679
C08514=1086.348,268.850,-81.389,176.196,23.056,153.679
C08515=1086.354,269.099,-81.417,176.199,23.059,153.679
C08516=1086.360,269.347,-81.445,176.202,23.062,153.680
C08517=1086.366,269.595,-81.474,176.205,23.065,153.680
C08518=1086.370,269.844,-81.503,176.207,23.068,153.680
C08519=1086.376,270.093,-81.531,176.210,23.071,153.680
C08520=1086.382,270.340,-81.560,176.213,23.075,153.681
C08521=1086.388,270.589,-81.588,176.216,23.078,153.681
C08522=1086.393,270.837,-81.616,176.218,23.081,153.681
C08523=1086.399,271.085,-81.646,176.221,23.084,153.682
C08524=1086.405,271.334,-81.674,176.224,23.087,153.682
C08525=1086.410,271.581,-81.703,176.227,23.090,153.682
C08526=1086.416,271.830,-81.731,176.230,23.093,153.682
C08527=1086.422,272.079,-81.759,176.232,23.096,153.683
C08528=1086.427,272.327,-81.789,176.235,23.099,153.683
C08529=1086.433,272.575,-81.817,176.238,23.102,153.683
C08530=1086.439,272.823,-81.846,176.241,23.106,153.684
C08531=1086.445,273.072,-81.874,176.244,23.108,153.684
C08532=1086.450,273.320,-81.904,176.247,23.112,153.684
C08533=1086.456,273.568,-81.932,176.250,23.115,153.684
C08534=1086.462,273.816,-81.961,176.253,23.118,153.685
C08535=1086.468,274.064,-81.990,176.256,23.121,153.685
C08536=1086.473,274.313,-82.018,176.258,23.124,153.685
C08537=1086.479,274.561,-82.047,176.261,23.128,153.686
C08538=1086.484,274.810,-82.076,176.264,23.131,153.686
C08539=1086.490,275.057,-82.105,176.267,23.134,153.686
C08540=1086.496,275.305,-82.134,176.270,23.137,153.687
C08541=1086.501,275.554,-82.163,176.272,23.140,153.687
C08542=1086.510,275.932,-82.207,176.276,23.145,153.687
C08543=1086.519,276.311,-82.251,176.281,23.150,153.688
C08544=1086.528,276.688,-82.295,176.286,23.154,153.688
C08545=1086.536,277.066,-82.338,176.290,23.159,153.689
C08546=1086.542,277.314,-82.368,176.292,23.162,153.689
C08547=1086.548,277.562,-82.397,176.295,23.165,153.689
C08548=1086.553,277.811,-82.427,176.298,23.169,153.689
C08549=1086.559,278.059,-82.455,176.301,23.172,153.690
C08550=1086.564,278.307,-82.484,176.304,23.175,153.690
C08551=1086.570,278.556,-82.513,176.307,23.179,153.690
C08552=1086.576,278.804,-82.543,176.309,23.181,153.691
C08553=1086.582,279.051,-82.572,176.312,23.184,153.691
C08554=1086.588,279.300,-82.601,176.316,23.188,153.691
C08555=1086.593,279.548,-82.630,176.319,23.191,153.692
C08556=1086.599,279.797,-82.659,176.321,23.195,153.692
C08557=1086.605,280.045,-82.688,176.324,23.198,153.692
C08558=1086.610,280.293,-82.718,176.327,23.200,153.693
C08559=1086.616,280.541,-82.747,176.330,23.204,153.693
C08560=1086.621,280.789,-82.776,176.333,23.207,153.693
C08561=1086.628,281.038,-82.805,176.336,23.210,153.693
C08562=1086.633,281.286,-82.835,176.339,23.214,153.694
C08563=1086.639,281.533,-82.864,176.342,23.217,153.694
C08564=1086.644,281.782,-82.893,176.344,23.220,153.694
C08565=1086.650,282.030,-82.923,176.347,23.223,153.695
C08566=1086.656,282.279,-82.952,176.350,23.226,153.695
C08567=1086.662,282.527,-82.982,176.353,23.230,153.695
C08568=1086.667,282.775,-83.011,176.356,23.233,153.696
C08569=1086.673,283.023,-83.040,176.359,23.236,153.696
C08570=1086.678,283.271,-83.070,176.362,23.240,153.696
C08571=1086.684,283.519,-83.100,176.364,23.242,153.697
C08572=1086.690,283.768,-83.130,176.367,23.245,153.697
C08573=1086.696,284.016,-83.159,176.370,23.249,153.697
C08574=1086.701,284.264,-83.188,176.373,23.252,153.698
C08575=1086.706,284.512,-83.217,176.376,23.255,153.698
C08576=1086.713,284.760,-83.247,176.379,23.259,153.698
C08577=1086.718,285.008,-83.276,176.382,23.262,153.699
C08578=1086.724,285.256,-83.307,176.385,23.265,153.699
C08579=1086.729,285.505,-83.336,176.387,23.268,153.699
C08580=1086.736,285.753,-83.365,176.390,23.272,153.700
C08581=1086.741,286.001,-83.395,176.393,23.275,153.700
C08582=1086.747,286.249,-83.425,176.396,23.278,153.700
C08583=1086.753,286.498,-83.455,176.399,23.282,153.701
C08584=1086.759,286.746,-83.484,176.402,23.285,153.701
C08585=1086.765,286.993,-83.514,176.405,23.288,153.701
C08586=1086.769,287.241,-83.543,176.408,23.292,153.702
C08587=1086.775,287.490,-83.573,176.411,23.295,153.702
C08588=1086.781,287.737,-83.603,176.413,23.298,153.702
C08589=1086.787,287.986,-83.633,176.416,23.301,153.703
C08590=1086.793,288.234,-83.662,176.419,23.305,153.703
C08591=1086.798,288.482,-83.692,176.422,23.308,153.703
C08592=1086.804,288.730,-83.722,176.425,23.311,153.703
C08593=1086.810,288.978,-83.752,176.428,23.315,153.704
C08594=1086.819,289.366,-83.799,176.433,23.320,153.704
C08595=1086.828,289.753,-83.846,176.437,23.325,153.705
C08596=1086.837,290.141,-83.892,176.441,23.330,153.706
C08597=1086.846,290.529,-83.940,176.446,23.335,153.706
C08598=1086.852,290.777,-83.969,176.449,23.338,153.706
C08599=1086.857,291.025,-84.000,176.452,23.342,153.707
C08600=1086.863,291.273,-84.029,176.455,23.345,153.707
C08601=1086.869,291.521,-84.059,176.458,23.349,153.707
C08602=1086.875,291.769,-84.090,176.461,23.352,153.708
C08603=1086.880,292.018,-84.119,176.464,23.355,153.708
C08604=1086.886,292.265,-84.150,176.467,23.359,153.708
C08605=1086.891,292.514,-84.179,176.470,23.362,153.709
C08606=1086.897,292.762,-84.210,176.473,23.365,153.709
C08607=1086.903,293.009,-84.240,176.476,23.369,153.710
C08608=1086.909,293.258,-84.270,176.479,23.372,153.710
C08609=1086.914,293.506,-84.300,176.482,23.376,153.710
C08610=1086.920,293.754,-84.330,176.484,23.379,153.711
C08611=1086.926,294.001,-84.361,176.487,23.382,153.711
C08612=1086.931,294.250,-84.390,176.490,23.385,153.711
C08613=1086.937,294.498,-84.421,176.493,23.389,153.712
C08614=1086.943,294.745,-84.451,176.496,23.392,153.712
C08615=1086.949,294.993,-84.482,176.499,23.396,153.712
C08616=1086.955,295.242,-84.513,176.502,23.399,153.713
C08617=1086.960,295.491,-84.542,176.505,23.403,153.713
C08618=1086.966,295.738,-84.573,176.508,23.406,153.713
C08619=1086.972,295.986,-84.603,176.511,23.409,153.714
C08620=1086.978,296.234,-84.634,176.514,23.413,153.714
C08621=1086.983,296.482,-84.664,176.516,23.416,153.714
C08622=1086.989,296.730,-84.694,176.520,23.419,153.715
C08623=1086.994,296.978,-84.725,176.522,23.423,153.715
C08624=1087.000,297.227,-84.755,176.525,23.427,153.716
C08625=1087.006,297.475,-84.786,176.528,23.430,153.716
C08626=1087.012,297.723,-84.816,176.531,23.433,153.716
C08627=1087.018,297.970,-84.846,176.534,23.437,153.717
C08628=1087.023,298.219,-84.877,176.537,23.440,153.717
C08629=1087.029,298.466,-84.908,176.540,23.444,153.717
C08630=1087.034,298.714,-84.938,176.543,23.447,153.718
C08631=1087.040,298.963,-84.969,176.546,23.451,153.718
C08632=1087.046,299.211,-85.000,176.549,23.454,153.719
C08633=1087.051,299.459,-85.030,176.552,23.458,153.719
C08634=1087.057,299.706,-85.062,176.555,23.461,153.719
C08635=1087.062,299.954,-85.092,176.558,23.465,153.720
C08636=1087.068,300.202,-85.123,176.561,23.468,153.720
C08637=1087.073,300.450,-85.154,176.564,23.472,153.721
C08638=1087.080,300.699,-85.185,176.567,23.476,153.721
C08639=1087.085,300.947,-85.215,176.569,23.479,153.721
C08640=1087.091,301.195,-85.246,176.572,23.483,153.722
C08641=1087.096,301.443,-85.276,176.575,23.486,153.722
C08642=1087.102,301.690,-85.308,176.578,23.490,153.722
C08643=1087.108,301.938,-85.338,176.581,23.493,153.723
C08644=1087.113,302.187,-85.369,176.584,23.497,153.723
C08645=1087.119,302.435,-85.400,176.587,23.500,153.724
C08646=1087.128,302.836,-85.450,176.591,23.506,153.724
C08647=1087.137,303.237,-85.501,176.597,23.512,153.725
C08648=1087.146,303.639,-85.550,176.601,23.517,153.726
C08649=1087.155,304.041,-85.601,176.606,23.524,153.726
C08650=1087.161,304.289,-85.631,176.609,23.527,153.727
C08651=1087.167,304.536,-85.663,176.612,23.530,153.727
C08652=1087.173,304.785,-85.694,176.615,23.534,153.727
C08653=1087.178,305.032,-85.725,176.618,23.538,153.728
C08654=1087.184,305.280,-85.756,176.621,23.541,153.728
C08655=1087.190,305.528,-85.788,176.624,23.545,153.729
C08656=1087.195,305.777,-85.819,176.627,23.548,153.729
C08657=1087.201,306.024,-85.849,176.630,23.552,153.730
C08658=1087.207,306.273,-85.881,176.633,23.555,153.730
C08659=1087.213,306.520,-85.911,176.636,23.559,153.730
C08660=1087.218,306.768,-85.943,176.638,23.562,153.731
C08661=1087.225,307.016,-85.974,176.641,23.566,153.731
C08662=1087.230,307.264,-86.005,176.645,23.570,153.732
C08663=1087.236,307.511,-86.037,176.648,23.574,153.732
C08664=1087.242,307.760,-86.068,176.651,23.577,153.732
C08665=1087.247,308.008,-86.099,176.654,23.581,153.733
C08666=1087.254,308.256,-86.130,176.657,23.585,153.733
C08667=1087.259,308.504,-86.162,176.660,23.588,153.734
C08668=1087.264,308.752,-86.193,176.663,23.592,153.734
C08669=1087.271,309.000,-86.224,176.666,23.595,153.734
C08670=1087.276,309.247,-86.256,176.668,23.599,153.735
C08671=1087.282,309.496,-86.287,176.672,23.602,153.735
C08672=1087.288,309.743,-86.318,176.674,23.606,153.736
C08673=1087.294,309.991,-86.350,176.677,23.609,153.736
C08674=1087.300,310.239,-86.382,176.680,23.613,153.736
C08675=1087.306,310.487,-86.413,176.683,23.617,153.737
C08676=1087.311,310.735,-86.444,176.687,23.621,153.737
C08677=1087.317,310.983,-86.476,176.690,23.624,153.738
C08678=1087.323,311.231,-86.507,176.693,23.628,153.738
C08679=1087.329,311.479,-86.539,176.696,23.632,153.739
C08680=1087.335,311.727,-86.570,176.699,23.635,153.739
C08681=1087.341,311.975,-86.602,176.702,23.639,153.739
C08682=1087.347,312.222,-86.633,176.705,23.642,153.740
C08683=1087.353,312.470,-86.666,176.707,23.646,153.740
C08684=1087.358,312.718,-86.696,176.710,23.650,153.741
C08685=1087.364,312.966,-86.728,176.713,23.653,153.741
C08686=1087.370,313.214,-86.760,176.716,23.657,153.742
C08687=1087.376,313.462,-86.792,176.720,23.661,153.742
C08688=1087.382,313.710,-86.824,176.723,23.664,153.742
C08689=1087.388,313.957,-86.855,176.726,23.668,153.743
C08690=1087.394,314.206,-86.887,176.729,23.672,153.743
C08691=1087.399,314.453,-86.918,176.732,23.675,153.744
C08692=1087.405,314.701,-86.950,176.735,23.679,153.744
C08693=1087.412,314.949,-86.982,176.737,23.683,153.745
C08694=1087.417,315.197,-87.013,176.740,23.687,153.745
C08695=1087.423,315.445,-87.046,176.743,23.690,153.745
C08696=1087.428,315.693,-87.078,176.747,23.695,153.746
C08697=1087.434,315.941,-87.110,176.750,23.698,153.746
C08698=1087.443,316.345,-87.162,176.754,23.704,153.747
C08699=1087.452,316.750,-87.214,176.759,23.711,153.748
C08700=1087.461,317.154,-87.266,176.764,23.717,153.749
C08701=1087.471,317.559,-87.319,176.769,23.724,153.750
C08702=1087.476,317.806,-87.351,176.772,23.727,153.750
C08703=1087.482,318.054,-87.383,176.775,23.731,153.751
C08704=1087.488,318.303,-87.415,176.778,23.735,153.751
C08705=1087.494,318.549,-87.447,176.781,23.739,153.751
C08706=1087.499,318.798,-87.480,176.784,23.743,153.752
C08707=1087.504,319.045,-87.511,176.786,23.747,153.752
C08708=1087.510,319.294,-87.543,176.790,23.751,153.753
C08709=1087.517,319.541,-87.576,176.793,23.755,153.753
C08710=1087.522,319.789,-87.608,176.796,23.758,153.754
C08711=1087.527,320.037,-87.640,176.799,23.762,153.754
C08712=1087.533,320.286,-87.672,176.802,23.766,153.755
C08713=1087.539,320.532,-87.705,176.804,23.770,153.755
C08714=1087.545,320.781,-87.737,176.808,23.774,153.756
C08715=1087.550,321.029,-87.769,176.811,23.778,153.756
C08716=1087.556,321.276,-87.802,176.814,23.782,153.757
C08717=1087.562,321.524,-87.834,176.817,23.786,153.757
C08718=1087.568,321.772,-87.867,176.820,23.789,153.758
C08719=1087.573,322.020,-87.899,176.822,23.794,153.758
C08720=1087.579,322.267,-87.932,176.826,23.798,153.759
C08721=1087.585,322.515,-87.964,176.829,23.802,153.759
C08722=1087.591,322.764,-87.996,176.832,23.806,153.760
C08723=1087.597,323.012,-88.029,176.835,23.809,153.760
C08724=1087.602,323.259,-88.061,176.837,23.813,153.761
C08725=1087.608,323.507,-88.093,176.841,23.818,153.761
C08726=1087.614,323.755,-88.127,176.844,23.821,153.762
C08727=1087.620,324.003,-88.159,176.847,23.826,153.762
C08728=1087.626,324.250,-88.191,176.850,23.829,153.763
C08729=1087.631,324.498,-88.224,176.853,23.833,153.763
C08730=1087.637,324.746,-88.257,176.856,23.838,153.764
C08731=1087.643,324.994,-88.289,176.859,23.841,153.764
C08732=1087.649,325.242,-88.322,176.862,23.845,153.765
C08733=1087.655,325.490,-88.355,176.865,23.849,153.765
C08734=1087.660,325.737,-88.386,176.868,23.853,153.766
C08735=1087.666,325.985,-88.420,176.871,23.857,153.766
C08736=1087.672,326.233,-88.452,176.874,23.862,153.767
C08737=1087.678,326.480,-88.485,176.877,23.865,153.767
C08738=1087.684,326.729,-88.518,176.880,23.869,153.768
C08739=1087.690,326.976,-88.550,176.883,23.873,153.768
C08740=1087.696,327.224,-88.583,176.887,23.877,153.769
C08741=1087.702,327.472,-88.617,176.889,23.881,153.769
C08742=1087.708,327.720,-88.649,176.892,23.885,153.770
C08743=1087.713,327.967,-88.682,176.895,23.889,153.771
C08744=1087.719,328.215,-88.714,176.899,23.893,153.771
C08745=1087.725,328.463,-88.748,176.902,23.898,153.772
C08746=1087.731,328.710,-88.780,176.904,23.902,153.772
C08747=1087.737,328.958,-88.812,176.907,23.906,153.773
C08748=1087.742,329.206,-88.846,176.911,23.910,153.773
C08749=1087.749,329.454,-88.879,176.914,23.914,153.774
C08750=1087.758,329.851,-88.932,176.919,23.920,153.775
C08751=1087.768,330.249,-88.985,176.924,23.927,153.775
C08752=1087.777,330.647,-89.037,176.928,23.933,153.776
C08753=1087.787,331.044,-89.091,176.933,23.940,153.777
C08754=1087.793,331.292,-89.124,176.937,23.944,153.778
C08755=1087.799,331.540,-89.157,176.939,23.948,153.778
C08756=1087.805,331.788,-89.190,176.942,23.952,153.779
C08757=1087.811,332.035,-89.223,176.945,23.956,153.779
C08758=1087.817,332.283,-89.257,176.949,23.961,153.780
C08759=1087.822,332.531,-89.290,176.952,23.965,153.780
C08760=1087.829,332.779,-89.323,176.954,23.969,153.781
C08761=1087.834,333.027,-89.356,176.958,23.973,153.781
C08762=1087.840,333.275,-89.389,176.961,23.978,153.782
C08763=1087.845,333.522,-89.423,176.963,23.982,153.783
C08764=1087.852,333.769,-89.456,176.966,23.986,153.783
C08765=1087.857,334.017,-89.489,176.970,23.991,153.784
C08766=1087.863,334.265,-89.523,176.973,23.995,153.784
C08767=1087.868,334.513,-89.556,176.975,23.999,153.785
C08768=1087.874,334.760,-89.590,176.979,24.004,153.786
C08769=1087.881,335.008,-89.623,176.982,24.008,153.786
C08770=1087.886,335.256,-89.656,176.985,24.012,153.787
C08771=1087.892,335.504,-89.690,176.988,24.016,153.787
C08772=1087.898,335.751,-89.724,176.991,24.021,153.788
C08773=1087.903,335.999,-89.757,176.994,24.025,153.789
C08774=1087.909,336.247,-89.790,176.998,24.029,153.789
C08775=1087.915,336.494,-89.824,177.000,24.034,153.790
C08776=1087.921,336.742,-89.857,177.003,24.038,153.790
C08777=1087.927,336.990,-89.891,177.007,24.042,153.791
C08778=1087.933,337.238,-89.925,177.010,24.046,153.791
C08779=1087.938,337.486,-89.958,177.012,24.051,153.792
C08780=1087.945,337.733,-89.992,177.016,24.055,153.793
C08781=1087.951,337.980,-90.025,177.019,24.059,153.793
C08782=1087.956,338.228,-90.059,177.021,24.064,153.794
C08783=1087.962,338.476,-90.092,177.025,24.068,153.794
C08784=1087.968,338.724,-90.127,177.028,24.073,153.795
C08785=1087.974,338.972,-90.160,177.031,24.077,153.796
C08786=1087.980,339.219,-90.194,177.034,24.082,153.796
C08787=1087.985,339.467,-90.228,177.037,24.086,153.797
C08788=1087.991,339.714,-90.262,177.040,24.091,153.798
C08789=1087.997,339.961,-90.296,177.043,24.095,153.798
C08790=1088.003,340.209,-90.329,177.046,24.099,153.799
C08791=1088.009,340.457,-90.363,177.049,24.104,153.800
C08792=1088.015,340.704,-90.397,177.052,24.108,153.800
C08793=1088.021,340.952,-90.431,177.056,24.113,153.801
C08794=1088.026,341.200,-90.465,177.059,24.117,153.801
C08795=1088.032,341.447,-90.499,177.061,24.122,153.802
C08796=1088.038,341.696,-90.533,177.065,24.127,153.803
C08797=1088.044,341.943,-90.567,177.068,24.131,153.803
C08798=1088.049,342.190,-90.601,177.071,24.136,153.804
C08799=1088.055,342.438,-90.635,177.074,24.140,153.805
C08800=1088.061,342.686,-90.669,177.077,24.144,153.805
C08801=1088.067,342.934,-90.703,177.080,24.149,153.806
C08802=1088.077,343.325,-90.757,177.085,24.156,153.807
C08803=1088.085,343.717,-90.811,177.090,24.163,153.808
C08804=1088.095,344.109,-90.865,177.095,24.170,153.809
C08805=1088.105,344.501,-90.920,177.100,24.178,153.810
C08806=1088.110,344.748,-90.954,177.103,24.182,153.811
C08807=1088.116,344.995,-90.988,177.106,24.187,153.811
C08808=1088.123,345.243,-91.022,177.109,24.192,153.812
C08809=1088.128,345.491,-91.057,177.112,24.196,153.813
C08810=1088.134,345.738,-91.091,177.115,24.201,153.813
C08811=1088.140,345.986,-91.125,177.118,24.205,153.814
C08812=1088.146,346.233,-91.159,177.121,24.210,153.815
C08813=1088.151,346.481,-91.194,177.124,24.215,153.816
C08814=1088.158,346.729,-91.228,177.127,24.220,153.816
C08815=1088.163,346.976,-91.262,177.130,24.224,153.817
C08816=1088.169,347.224,-91.297,177.134,24.229,153.818
C08817=1088.175,347.472,-91.331,177.136,24.234,153.818
C08818=1088.181,347.719,-91.365,177.140,24.239,153.819
C08819=1088.186,347.967,-91.400,177.143,24.243,153.820
C08820=1088.192,348.215,-91.435,177.146,24.248,153.820
C08821=1088.198,348.462,-91.470,177.149,24.253,153.821
C08822=1088.204,348.709,-91.504,177.152,24.258,153.822
C08823=1088.210,348.957,-91.538,177.155,24.262,153.822
C08824=1088.215,349.204,-91.573,177.159,24.267,153.823
C08825=1088.222,349.452,-91.608,177.161,24.272,153.824
C08826=1088.227,349.699,-91.643,177.165,24.277,153.825
C08827=1088.233,349.947,-91.677,177.167,24.282,153.825
C08828=1088.240,350.195,-91.711,177.171,24.286,153.826
C08829=1088.245,350.442,-91.747,177.174,24.291,153.827
C08830=1088.251,350.690,-91.781,177.177,24.296,153.828
C08831=1088.257,350.937,-91.816,177.180,24.301,153.828
C08832=1088.263,351.185,-91.851,177.183,24.306,153.829
C08833=1088.268,351.432,-91.885,177.186,24.311,153.830
C08834=1088.275,351.679,-91.920,177.189,24.316,153.830
C08835=1088.280,351.927,-91.955,177.192,24.320,153.831
C08836=1088.287,352.174,-91.990,177.196,24.325,153.832
C08837=1088.292,352.422,-92.025,177.198,24.330,153.833
C08838=1088.298,352.669,-92.060,177.202,24.335,153.833
C08839=1088.304,352.917,-92.095,177.204,24.340,153.834
C08840=1088.310,353.164,-92.130,177.208,24.345,153.835
C08841=1088.316,353.412,-92.165,177.211,24.350,153.836
C08842=1088.322,353.659,-92.199,177.214,24.354,153.836
C08843=1088.328,353.907,-92.234,177.217,24.359,153.837
C08844=1088.333,354.154,-92.270,177.220,24.365,153.838
C08845=1088.340,354.402,-92.304,177.224,24.370,153.839
C08846=1088.345,354.649,-92.340,177.226,24.375,153.839
C08847=1088.351,354.897,-92.375,177.230,24.380,153.840
C08848=1088.357,355.144,-92.409,177.232,24.384,153.841
C08849=1088.363,355.392,-92.445,177.236,24.390,153.842
C08850=1088.369,355.639,-92.480,177.238,24.395,153.843
C08851=1088.374,355.887,-92.515,177.242,24.400,153.843
C08852=1088.381,356.134,-92.551,177.245,24.405,153.844
C08853=1088.387,356.381,-92.586,177.248,24.410,153.845
C08854=1088.396,356.776,-92.642,177.253,24.418,153.846
C08855=1088.405,357.170,-92.698,177.258,24.426,153.847
C08856=1088.415,357.564,-92.755,177.263,24.434,153.849
C08857=1088.424,357.959,-92.810,177.268,24.443,153.850
C08858=1088.430,358.207,-92.846,177.271,24.447,153.851
C08859=1088.436,358.455,-92.882,177.275,24.453,153.852
C08860=1088.442,358.701,-92.917,177.277,24.458,153.852
C08861=1088.448,358.949,-92.952,177.281,24.463,153.853
C08862=1088.454,359.197,-92.988,177.283,24.468,153.854
C08863=1088.460,359.444,-93.023,177.287,24.473,153.855
C08864=1088.466,359.691,-93.059,177.290,24.479,153.856
C08865=1088.473,359.939,-93.094,177.293,24.484,153.856
C08866=1088.478,360.186,-93.130,177.296,24.489,153.857
C08867=1088.484,360.433,-93.165,177.299,24.494,153.858
C08868=1088.490,360.681,-93.201,177.302,24.500,153.859
C08869=1088.496,360.928,-93.237,177.305,24.505,153.860
C08870=1088.502,361.176,-93.272,177.308,24.510,153.861
C08871=1088.508,361.423,-93.308,177.312,24.515,153.862
C08872=1088.513,361.670,-93.344,177.315,24.521,153.862
C08873=1088.519,361.917,-93.380,177.317,24.526,153.863
C08874=1088.525,362.165,-93.416,177.321,24.531,153.864
C08875=1088.531,362.412,-93.451,177.324,24.537,153.865
C08876=1088.537,362.660,-93.487,177.327,24.542,153.866
C08877=1088.543,362.907,-93.523,177.330,24.547,153.867
C08878=1088.549,363.154,-93.559,177.334,24.553,153.867
C08879=1088.555,363.401,-93.594,177.336,24.558,153.868
C08880=1088.561,363.649,-93.630,177.340,24.563,153.869
C08881=1088.567,363.896,-93.666,177.343,24.569,153.870
C08882=1088.573,364.144,-93.702,177.346,24.574,153.871
C08883=1088.578,364.391,-93.737,177.349,24.580,153.872
C08884=1088.585,364.638,-93.774,177.352,24.585,153.873
C08885=1088.591,364.885,-93.810,177.355,24.591,153.874
C08886=1088.597,365.133,-93.845,177.358,24.596,153.875
C08887=1088.603,365.380,-93.882,177.362,24.602,153.875
C08888=1088.609,365.627,-93.917,177.364,24.607,153.876
C08889=1088.615,365.874,-93.954,177.367,24.613,153.877
C08890=1088.620,366.122,-93.990,177.371,24.618,153.878
C08891=1088.627,366.369,-94.026,177.374,24.624,153.879
C08892=1088.632,366.616,-94.062,177.377,24.629,153.880
C08893=1088.638,366.863,-94.098,177.380,24.635,153.881
C08894=1088.644,367.111,-94.134,177.383,24.641,153.882
C08895=1088.650,367.358,-94.171,177.386,24.646,153.883
C08896=1088.656,367.605,-94.207,177.389,24.652,153.884
C08897=1088.662,367.852,-94.243,177.393,24.658,153.885
C08898=1088.668,368.099,-94.279,177.396,24.663,153.886
C08899=1088.673,368.347,-94.316,177.398,24.669,153.887
C08900=1088.680,368.594,-94.352,177.402,24.674,153.888
C08901=1088.686,368.841,-94.388,177.405,24.680,153.889
C08902=1088.691,369.089,-94.425,177.408,24.686,153.889
C08903=1088.698,369.336,-94.461,177.411,24.691,153.890
C08904=1088.703,369.583,-94.497,177.414,24.697,153.891
C08905=1088.709,369.830,-94.534,177.418,24.703,153.892
C08906=1088.719,370.240,-94.595,177.423,24.712,153.894
C08907=1088.729,370.650,-94.655,177.428,24.722,153.896
C08908=1088.739,371.060,-94.716,177.433,24.731,153.897
C08909=1088.750,371.471,-94.776,177.438,24.741,153.899
C08910=1088.755,371.717,-94.812,177.441,24.747,153.900
C08911=1088.761,371.965,-94.849,177.444,24.753,153.901
C08912=1088.767,372.212,-94.886,177.448,24.759,153.902
C08913=1088.773,372.459,-94.923,177.451,24.764,153.903
C08914=1088.779,372.706,-94.959,177.453,24.770,153.904
C08915=1088.786,372.953,-94.996,177.457,24.776,153.905
C08916=1088.791,373.201,-95.033,177.460,24.782,153.906
C08917=1088.798,373.448,-95.069,177.463,24.788,153.907
C08918=1088.804,373.695,-95.106,177.467,24.794,153.908
C08919=1088.810,373.942,-95.143,177.469,24.800,153.909
C08920=1088.816,374.190,-95.180,177.472,24.805,153.910
C08921=1088.822,374.437,-95.217,177.476,24.812,153.911
C08922=1088.827,374.684,-95.253,177.479,24.818,153.912
C08923=1088.833,374.931,-95.290,177.482,24.824,153.913
C08924=1088.839,375.178,-95.327,177.486,24.830,153.914
C08925=1088.846,375.425,-95.364,177.488,24.836,153.915
C08926=1088.851,375.672,-95.401,177.491,24.842,153.916
C08927=1088.857,375.919,-95.438,177.494,24.848,153.917
C08928=1088.864,376.167,-95.475,177.498,24.854,153.918
C08929=1088.870,376.414,-95.513,177.501,24.860,153.919
C08930=1088.875,376.661,-95.550,177.504,24.866,153.920
C08931=1088.882,376.908,-95.586,177.507,24.872,153.921
C08932=1088.887,377.155,-95.624,177.510,24.878,153.922
C08933=1088.893,377.402,-95.661,177.513,24.884,153.923
C08934=1088.899,377.650,-95.697,177.516,24.891,153.924
C08935=1088.905,377.896,-95.735,177.520,24.897,153.926
C08936=1088.911,378.144,-95.772,177.523,24.903,153.927
C08937=1088.917,378.391,-95.809,177.526,24.909,153.928
C08938=1088.923,378.637,-95.846,177.529,24.916,153.929
C08939=1088.929,378.885,-95.883,177.532,24.922,153.930
C08940=1088.936,379.132,-95.921,177.535,24.928,153.931
C08941=1088.942,379.379,-95.958,177.538,24.934,153.932
C08942=1088.948,379.626,-95.996,177.541,24.940,153.933
C08943=1088.953,379.873,-96.033,177.545,24.947,153.934
C08944=1088.960,380.120,-96.070,177.548,24.953,153.936
C08945=1088.966,380.367,-96.108,177.551,24.959,153.937
C08946=1088.972,380.615,-96.145,177.554,24.966,153.938
C08947=1088.978,380.861,-96.183,177.557,24.972,153.939
C08948=1088.984,381.108,-96.220,177.561,24.979,153.940
C08949=1088.990,381.355,-96.257,177.564,24.985,153.941
C08950=1088.996,381.602,-96.295,177.567,24.991,153.942
C08951=1089.002,381.849,-96.333,177.569,24.997,153.943
C08952=1089.009,382.096,-96.369,177.572,25.004,153.945
C08953=1089.015,382.343,-96.407,177.576,25.011,153.946
C08954=1089.021,382.590,-96.445,177.579,25.017,153.947
C08955=1089.027,382.837,-96.483,177.582,25.023,153.948
C08956=1089.033,383.085,-96.520,177.585,25.030,153.949
C08957=1089.039,383.331,-96.558,177.588,25.037,153.950
C08958=1089.044,383.550,-96.591,177.592,25.042,153.951
C08959=1089.049,383.769,-96.625,177.594,25.048,153.952
C08960=1089.055,383.988,-96.658,177.596,25.054,153.954
C08961=1089.060,384.207,-96.691,177.600,25.060,153.955
C08962=1089.065,384.426,-96.725,177.602,25.066,153.956
C08963=1089.071,384.645,-96.759,177.606,25.072,153.957
C08964=1089.076,384.864,-96.793,177.608,25.078,153.958
C08965=1089.081,385.083,-96.826,177.611,25.084,153.959
C08966=1089.087,385.330,-96.864,177.614,25.090,153.960
C08967=1089.093,385.577,-96.902,177.618,25.097,153.961
C08968=1089.099,385.823,-96.939,177.621,25.104,153.962
C08969=1089.106,386.071,-96.977,177.624,25.111,153.964
C08970=1089.112,386.318,-97.015,177.627,25.117,153.965
C08971=1089.118,386.564,-97.053,177.630,25.124,153.966
C08972=1089.124,386.812,-97.091,177.633,25.131,153.967
C08973=1089.129,387.059,-97.129,177.636,25.138,153.969
C08974=1089.135,387.305,-97.168,177.639,25.144,153.970
C08975=1089.142,387.552,-97.206,177.643,25.151,153.971
C08976=1089.148,387.799,-97.244,177.646,25.158,153.973
C08977=1089.154,388.046,-97.282,177.649,25.165,153.974
C08978=1089.160,388.293,-97.320,177.652,25.172,153.975
C08979=1089.166,388.540,-97.358,177.655,25.179,153.976
C08980=1089.172,388.786,-97.396,177.658,25.186,153.978
C08981=1089.178,389.034,-97.435,177.661,25.192,153.979
C08982=1089.184,389.280,-97.473,177.664,25.199,153.980
C08983=1089.191,389.528,-97.511,177.667,25.206,153.981
C08984=1089.197,389.774,-97.549,177.670,25.213,153.983
C08985=1089.204,390.021,-97.588,177.674,25.221,153.984
C08986=1089.210,390.268,-97.626,177.678,25.227,153.985
C08987=1089.216,390.515,-97.665,177.681,25.234,153.987
C08988=1089.221,390.762,-97.703,177.684,25.241,153.988
C08989=1089.228,391.009,-97.741,177.687,25.248,153.989
C08990=1089.234,391.255,-97.779,177.690,25.255,153.990
C08991=1089.241,391.503,-97.817,177.693,25.262,153.992
C08992=1089.246,391.749,-97.857,177.696,25.269,153.993
C08993=1089.253,391.997,-97.895,177.699,25.276,153.994
C08994=1089.259,392.243,-97.933,177.703,25.284,153.996
C08995=1089.265,392.490,-97.973,177.706,25.291,153.997
C08996=1089.271,392.737,-98.010,177.709,25.298,153.999
C08997=1089.278,392.984,-98.049,177.712,25.305,154.000
C08998=1089.283,393.231,-98.088,177.715,25.313,154.001
C08999=1089.290,393.477,-98.126,177.718,25.320,154.003
C09000=1089.296,393.725,-98.166,177.721,25.327,154.004
C09001=1089.302,393.971,-98.204,177.725,25.335,154.005
C09002=1089.308,394.218,-98.243,177.728,25.342,154.007
C09003=1089.314,394.465,-98.281,177.731,25.349,154.008
C09004=1089.320,394.712,-98.321,177.734,25.357,154.010
C09005=1089.327,394.959,-98.359,177.737,25.364,154.011
C09006=1089.333,395.205,-98.397,177.740,25.371,154.012
C09007=1089.339,395.452,-98.437,177.744,25.379,154.014
C09008=1089.344,395.699,-98.476,177.747,25.386,154.015
C09009=1089.351,395.946,-98.515,177.750,25.394,154.017
C09010=1089.357,396.193,-98.554,177.753,25.401,154.018
C09011=1089.363,396.440,-98.592,177.756,25.408,154.019
C09012=1089.369,396.687,-98.631,177.760,25.416,154.021
C09013=1089.375,396.934,-98.671,177.763,25.424,154.022
C09014=1089.381,397.159,-98.707,177.765,25.431,154.024
C09015=1089.387,397.384,-98.742,177.768,25.438,154.025
C09016=1089.392,397.611,-98.778,177.771,25.445,154.026
C09017=1089.398,397.836,-98.814,177.774,25.452,154.028
C09018=1089.404,398.061,-98.849,177.777,25.459,154.029
C09019=1089.409,398.287,-98.886,177.780,25.465,154.030
C09020=1089.415,398.513,-98.921,177.783,25.473,154.032
C09021=1089.421,398.739,-98.957,177.786,25.480,154.033
C09022=1089.427,398.985,-98.996,177.789,25.488,154.035
C09023=1089.433,399.232,-99.035,177.792,25.495,154.036
C09024=1089.440,399.479,-99.075,177.796,25.503,154.038
C09025=1089.446,399.726,-99.114,177.798,25.511,154.039
C09026=1089.452,399.973,-99.154,177.801,25.518,154.041
C09027=1089.457,400.219,-99.193,177.805,25.527,154.042
C09028=1089.463,400.466,-99.232,177.808,25.535,154.044
C09029=1089.470,400.713,-99.272,177.811,25.542,154.045
C09030=1089.477,400.960,-99.311,177.814,25.550,154.047
C09031=1089.483,401.207,-99.351,177.818,25.559,154.048
C09032=1089.489,401.453,-99.390,177.821,25.566,154.050
C09033=1089.495,401.700,-99.430,177.824,25.574,154.052
C09034=1089.501,401.947,-99.469,177.827,25.582,154.053
C09035=1089.507,402.193,-99.509,177.830,25.590,154.055
C09036=1089.513,402.441,-99.549,177.833,25.598,154.056
C09037=1089.520,402.687,-99.588,177.837,25.607,154.058
C09038=1089.526,402.934,-99.628,177.840,25.615,154.059
C09039=1089.532,403.181,-99.667,177.843,25.623,154.061
C09040=1089.539,403.428,-99.707,177.847,25.631,154.063
C09041=1089.544,403.674,-99.746,177.849,25.639,154.064
C09042=1089.551,403.921,-99.787,177.853,25.647,154.066
C09043=1089.557,404.168,-99.826,177.856,25.656,154.068
C09044=1089.563,404.414,-99.866,177.859,25.663,154.069
C09045=1089.569,404.661,-99.906,177.863,25.672,154.071
C09046=1089.576,404.908,-99.946,177.865,25.680,154.072
C09047=1089.582,405.154,-99.986,177.869,25.689,154.074
C09048=1089.588,405.401,-100.026,177.872,25.697,154.076
C09049=1089.594,405.648,-100.065,177.875,25.705,154.077
C09050=1089.601,405.894,-100.106,177.879,25.714,154.079
C09051=1089.607,406.141,-100.146,177.881,25.722,154.081
C09052=1089.613,406.388,-100.185,177.885,25.730,154.082
C09053=1089.620,406.635,-100.225,177.888,25.739,154.084
C09054=1089.625,406.881,-100.266,177.892,25.748,154.086
C09055=1089.632,407.128,-100.306,177.895,25.756,154.088
C09056=1089.638,407.375,-100.346,177.898,25.765,154.089
C09057=1089.644,407.621,-100.386,177.901,25.773,154.091
C09058=1089.651,407.868,-100.427,177.905,25.782,154.093
C09059=1089.657,408.115,-100.466,177.908,25.790,154.094
C09060=1089.662,408.362,-100.507,177.911,25.799,154.096
C09061=1089.669,408.608,-100.547,177.914,25.808,154.098
C09062=1089.676,408.855,-100.587,177.918,25.817,154.100
C09063=1089.681,409.102,-100.628,177.920,25.825,154.101
C09064=1089.688,409.349,-100.668,177.924,25.834,154.103
C09065=1089.694,409.595,-100.708,177.927,25.843,154.105
C09066=1089.700,409.841,-100.750,177.931,25.852,154.107
C09067=1089.707,410.088,-100.790,177.934,25.861,154.109
C09068=1089.713,410.334,-100.830,177.937,25.869,154.110
C09069=1089.719,410.581,-100.871,177.941,25.879,154.112
C09070=1089.724,410.807,-100.908,177.944,25.887,154.114
C09071=1089.730,411.033,-100.945,177.946,25.895,154.115
C09072=1089.737,411.260,-100.982,177.949,25.903,154.117
C09073=1089.742,411.486,-101.020,177.952,25.912,154.119
C09074=1089.748,411.713,-101.057,177.955,25.919,154.120
C09075=1089.754,411.938,-101.094,177.959,25.928,154.122
C09076=1089.759,412.165,-101.131,177.962,25.937,154.124
C09077=1089.765,412.391,-101.169,177.965,25.945,154.126
C09078=1089.772,412.637,-101.209,177.967,25.954,154.127
C09079=1089.778,412.884,-101.251,177.971,25.963,154.129
C09080=1089.784,413.131,-101.291,177.975,25.972,154.131
C09081=1089.790,413.377,-101.332,177.977,25.981,154.133
C09082=1089.797,413.624,-101.373,177.981,25.991,154.135
C09083=1089.803,413.871,-101.414,177.985,26.000,154.137
C09084=1089.810,414.117,-101.454,177.988,26.009,154.139
C09085=1089.816,414.363,-101.495,177.991,26.018,154.141
C09086=1089.823,414.610,-101.536,177.994,26.028,154.143
C09087=1089.829,414.857,-101.577,177.998,26.037,154.144
C09088=1089.835,415.103,-101.618,178.001,26.046,154.146
C09089=1089.842,415.349,-101.659,178.004,26.056,154.148
C09090=1089.848,415.596,-101.700,178.008,26.065,154.150
C09091=1089.855,415.843,-101.741,178.012,26.075,154.152
C09092=1089.861,416.089,-101.783,178.014,26.084,154.154
C09093=1089.868,416.336,-101.823,178.018,26.094,154.156
C09094=1089.874,416.582,-101.865,178.021,26.103,154.158
C09095=1089.880,416.829,-101.906,178.025,26.113,154.160
